// TwinCAT 3 PLC project RunTimeRoofControl
// Title: STELLA DachSteuerung
// Company: Leibniz Institut fuer Astrophysik Potsdam
// Author: J.Weingrill
// ProgramVersion: 3.1.4020.10
// libraries:
//   Tc2_Math, * (Beckhoff Automation GmbH)
//   Tc2_Standard, * (Beckhoff Automation GmbH)
//   Tc2_System, * (Beckhoff Automation GmbH)
//   Tc2_Utilities, * (Beckhoff Automation GmbH)
//   Tc3_IotBase, * (Beckhoff Automation GmbH)
//   Tc3_Module, * (Beckhoff Automation GmbH)
// project tree:
//   DUTs/ E_ErrorFlag.TcDUT, E_RoofCommand.TcDUT, E_RoofMode.TcDUT, E_RoofStatus.TcDUT
//   GVLs/ GVL_Environment.TcGVL, GVL_Infrastructure.TcGVL, GVL_Panel.TcGVL, GVL_Roof.TcGVL
//   / PlcTask.TcTTO
//   POUs/ Auxiliary.TcPOU, CalibrationUnit.TcPOU, Chamber.TcPOU, DehumidifierControl.TcPOU, Logging.TcPOU, MAIN.TcPOU, Environment.TcPOU
//   POUs/Function Blocks/ FB_AstroClock.TcPOU (not stored), FB_BLINK.TcPOU, FB_Dust.TcPOU (not stored), FB_EQ2HOR2.TcPOU (not stored), FB_EventLog.TcPOU, FB_Kalman1D.TcPOU, FB_MQTTCommunication.TcPOU, FB_PRECESS3.TcPOU, FB_RoofControl.TcPOU, FB_StatusLamp.TcPOU, FB_SUNPOS.TcPOU (not stored), FB_TimeAverage.TcPOU (not stored), InfluxMessage.TcPOU (not stored), LIGHT_BUTTON.TcPOU, TIMER.TcPOU
//   POUs/Functions/ APPEND.TcPOU (not stored), ATAN2.TcPOU (not stored), CT2LST.TcPOU (not stored), DateTime2JD.TcPOU (not stored), F_RainConversion.TcPOU (not stored), F_Y.TcPOU, Refraction.TcPOU (not stored), RoofStatus_TO_String.TcPOU
// real-time tasks:
//   TASK PlcTask: cycle T#10ms, priority 20, ADS port 350
// I/O:
//   DEVICE Device 1 (EtherCAT), AmsNetId 5.40.71.146.2.1
//     Term 1 (EK1200) [EK1200-5000 EtherCAT Power supply (2A E-Bus)]
//       Modul1 (EL2008) [EL2008 8Ch. Dig. Output 24V, 0.5A]
//       Modul2 (EL1008) [EL1008 8Ch. Dig. Input 24V, 3ms]
//       Modul3 (EL1008) [EL1008 8Ch. Dig. Input 24V, 3ms]
//       Modul4 (EL2008) [EL2008 8Ch. Dig. Output 24V, 0.5A]
//       Modul5 (EL1008) [EL1008 8Ch. Dig. Input 24V, 3ms]
//       Modul6 (EL1008) [EL1008 8Ch. Dig. Input 24V, 3ms] // Überstromkette Dach2
//       Modul7 (EL1008) [EL1008 8Ch. Dig. Input 24V, 3ms] // Panel
//       Modul8 (EL3068) [EL3068 8Ch. Ana. Input 0-10V] // Umweltsensoren innen
//       Modul9 (EL2008) [EL2008 8Ch. Dig. Output 24V, 0.5A]
//       Term 21 (EL9410) [EL9410 E-Bus Power Supplier  (Diagnostics)]
//       Modul10 (EL1024) [EL1024 4Ch. Dig. Input 24V, Type 2, 3ms] // Lichtschalter
//       Modul11 (EL3024) [EL3024 4Ch. Ana. Input 4-20mA DIFF]
//       Term 31 (EK1521) [EK1521 1 port EtherCAT junction (FX-MultiMode)]
//         WeatherStation1 (EK1501) [EK1501 EtherCAT Coupler (2A E-Bus, FX-MultiMode, ID switch)]
//           Term 33 (EL3068) [EL3068 8Ch. Ana. Input 0-10V]
//           Term 34 (EL1024) [EL1024 4Ch. Dig. Input 24V, Type 2, 3ms]
//           Term 35 (EL3024) [EL3024 4Ch. Ana. Input 4-20mA DIFF] // 1 Humidity,Temperature
//           Term 44 (EL6021) [EL6021 Interface (RS422/485)]
//           Term 41 (EL9011) [EL9011 End Terminal]
//       Term 36 (EK1521) [EK1521 1 port EtherCAT junction (FX-MultiMode)]
//         WeatherStation2 (EK1501) [EK1501 EtherCAT Coupler (2A E-Bus, FX-MultiMode, ID switch)]
//           Term 38 (EL3068) [EL3068 8Ch. Ana. Input 0-10V]
//           Term 39 (EL1024) [EL1024 4Ch. Dig. Input 24V, Type 2, 3ms]
//           Term 40 (EL3024) [EL3024 4Ch. Ana. Input 4-20mA DIFF]
//           Term 53 (EL6021) [EL6021 Interface (RS422/485)]
//           Term 42 (EL9011) [EL9011 End Terminal]
//       Term 56 (EK1521) [EK1521 1 port EtherCAT junction (FX-MultiMode)]
//         CalibrationUnit (EK1501) [EK1501 EtherCAT Coupler (2A E-Bus, FX-MultiMode, ID switch)]
//           Term 68 (EL1008) [EL1008 8Ch. Dig. Input 24V, 3ms]
//           Term 60 (EL2008) [EL2008 8Ch. Dig. Output 24V, 0.5A]
//           Term 61 (EL3164) [EL3164 4Ch. Ana. Input 0-10V]
//           Term 62 (EL3052) [EL3052 2Ch. Ana. Input 4-20mA]
//           Term 63 (EL3202-0010) [EL3202-0010 2Ch. Ana. Input PT100 (RTD), High Precision]
//           Term 64 (EL3202-0010) [EL3202-0010 2Ch. Ana. Input PT100 (RTD), High Precision]
//           Term 65 (EL3202-0010) [EL3202-0010 2Ch. Ana. Input PT100 (RTD), High Precision]
//           Term 76 (EK1110) [EK1110 EtherCAT extension]
//         Spectrograph Room (EK1100) [EK1100 EtherCAT Coupler (2A E-Bus)]
//           Term 79 (EL3202-0010) [EL3202-0010 2Ch. Ana. Input PT100 (RTD), High Precision]
//           Term 80 (EL3202-0010) [EL3202-0010 2Ch. Ana. Input PT100 (RTD), High Precision]
//           Term 81 (EL3202-0010) [EL3202-0010 2Ch. Ana. Input PT100 (RTD), High Precision]
//           Term 82 (EL3054) [EL3054 4Ch. Ana. Input 4-20mA]
//           Term 88 (EL9011) [EL9011 End Terminal]
//       Term 71 (EL9011) [EL9011 End Terminal]
//       Term 47 (EL9505) [EL9505 Power supply terminal 5V]
//       Term 48 (EL1124) [EL1124 4Ch. Dig. Input 5V, 10µs, Sensor Power]
//       Term 58 (EL1008) [EL1008 8Ch. Dig. Input 24V, 3ms]
//       Term 51 (EL9011) [EL9011 End Terminal]
//   DEVICE Device 3 (EtherCAT Automation Protocol) (disabled), AmsNetId 5.40.71.146.4.1
// variable links:
//   RunTimeRoofControl/RunTimeRoofControl Instance <-> Device 1 (EtherCAT)/Term 1 (EK1200)/Modul1 (EL2008)
//     PlcTask Outputs/GVL_Roof.ODach1Schnell <-> Channel 7/GVL_Roof.ODach1Schnell
//     PlcTask Outputs/GVL_Roof.ODach1auf <-> Channel 1/GVL_Roof.ODach1auf
//     PlcTask Outputs/GVL_Roof.ODach1zu <-> Channel 2/GVL_Roof.ODach1zu
//     PlcTask Outputs/GVL_Roof.ORiegel11auf <-> Channel 3/GVL_Roof.ORiegel11auf
//     PlcTask Outputs/GVL_Roof.ORiegel21auf <-> Channel 4/GVL_Roof.ORiegel21auf
//     PlcTask Outputs/GVL_Roof.ORiegel11zu <-> Channel 5/GVL_Roof.ORiegel11zu
//     PlcTask Outputs/GVL_Roof.ORiegel21zu <-> Channel 6/GVL_Roof.ORiegel21zu
//   RunTimeRoofControl/RunTimeRoofControl Instance <-> Device 1 (EtherCAT)/Term 1 (EK1200)/Modul10 (EL1024)
//     PlcTask Inputs/GVL_Environment.LightSwitch <-> Channel 1/Environment.LightSwitch
//   RunTimeRoofControl/RunTimeRoofControl Instance <-> Device 1 (EtherCAT)/Term 1 (EK1200)/Modul11 (EL3024)
//     PlcTask Inputs/GVL_Environment.DustSensorError <-> AI Standard Channel 1/Status/Error
//     PlcTask Inputs/GVL_Environment.rawDust <-> AI Standard Channel 1/Dust
//   RunTimeRoofControl/RunTimeRoofControl Instance <-> Device 1 (EtherCAT)/Term 1 (EK1200)/Modul2 (EL1008)
//     PlcTask Inputs/GVL_Roof.IDach1auf <-> Channel 1/GVL_Roof.IDach1auf
//     PlcTask Inputs/GVL_Roof.IDach1auf2 <-> Channel 2/GVL_Roof.IDach1auf2
//     PlcTask Inputs/GVL_Roof.IDach1zu <-> Channel 7/GVL_Roof.IDach1zu
//     PlcTask Inputs/GVL_Roof.IDach1zu2 <-> Channel 8/GVL_Roof.IDach1zu2
//     PlcTask Inputs/GVL_Roof.IRiegel11auf <-> Channel 3/GVL_Roof.IRiegel11auf
//     PlcTask Inputs/GVL_Roof.IRiegel21auf <-> Channel 4/GVL_Roof.IRiegel21auf
//     PlcTask Inputs/GVL_Roof.IRiegel11zu <-> Channel 5/GVL_Roof.IRiegel11zu
//     PlcTask Inputs/GVL_Roof.IRiegel21zu <-> Channel 6/GVL_Roof.IRiegel21zu
//   RunTimeRoofControl/RunTimeRoofControl Instance <-> Device 1 (EtherCAT)/Term 1 (EK1200)/Modul3 (EL1008)
//     PlcTask Inputs/GVL_Roof.IMotorschutz{11..16} <-> Channel {1..6}/GVL_Roof.IMotorschutz{11..16}  (6 links)
//   RunTimeRoofControl/RunTimeRoofControl Instance <-> Device 1 (EtherCAT)/Term 1 (EK1200)/Modul4 (EL2008)
//     PlcTask Outputs/GVL_Roof.ODach2Schnell <-> Channel 7/GVL_Roof.ODach2Schnell
//     PlcTask Outputs/GVL_Roof.ODach2auf <-> Channel 1/GVL_Roof.ODach2auf
//     PlcTask Outputs/GVL_Roof.ODach2zu <-> Channel 2/GVL_Roof.ODach2zu
//     PlcTask Outputs/GVL_Roof.ORiegel12auf <-> Channel 3/GVL_Roof.ORiegel12auf
//     PlcTask Outputs/GVL_Roof.ORiegel22auf <-> Channel 4/GVL_Roof.ORiegel22auf
//     PlcTask Outputs/GVL_Roof.ORiegel12zu <-> Channel 5/GVL_Roof.ORiegel12zu
//     PlcTask Outputs/GVL_Roof.ORiegel22zu <-> Channel 6/GVL_Roof.ORiegel22zu
//   RunTimeRoofControl/RunTimeRoofControl Instance <-> Device 1 (EtherCAT)/Term 1 (EK1200)/Modul5 (EL1008)
//     PlcTask Inputs/GVL_Roof.IDach2auf <-> Channel 1/GVL_Roof.IDach2auf
//     PlcTask Inputs/GVL_Roof.IDach2auf2 <-> Channel 2/GVL_Roof.IDach2auf2
//     PlcTask Inputs/GVL_Roof.IDach2zu <-> Channel 7/GVL_Roof.IDach2zu
//     PlcTask Inputs/GVL_Roof.IDach2zu2 <-> Channel 8/GVL_Roof.IDach2zu2
//     PlcTask Inputs/GVL_Roof.IRiegel12auf <-> Channel 3/GVL_Roof.IRiegel12auf
//     PlcTask Inputs/GVL_Roof.IRiegel22auf <-> Channel 4/GVL_Roof.IRiegel22auf
//     PlcTask Inputs/GVL_Roof.IRiegel12zu <-> Channel 5/GVL_Roof.IRiegel12zu
//     PlcTask Inputs/GVL_Roof.IRiegel22zu <-> Channel 6/GVL_Roof.IRiegel22zu
//   RunTimeRoofControl/RunTimeRoofControl Instance <-> Device 1 (EtherCAT)/Term 1 (EK1200)/Modul6 (EL1008)
//     PlcTask Inputs/GVL_Roof.IMotorschutz{21..26} <-> Channel {1..6}/GVL_Roof.IMotorschutz{21..26}  (6 links)
//   RunTimeRoofControl/RunTimeRoofControl Instance <-> Device 1 (EtherCAT)/Term 1 (EK1200)/Modul7 (EL1008)
//     PlcTask Inputs/GVL_Panel.ILeftCloseswitch <-> Channel 3/GVL_Panel.ILeftCloseswitch
//     PlcTask Inputs/GVL_Panel.ILeftOpenswitch <-> Channel 2/GVL_Panel.ILeftOpenswitch
//     PlcTask Inputs/GVL_Panel.IManualSwitch <-> Channel 1/GVL_Panel.IManualSwitch
//     PlcTask Inputs/GVL_Panel.IRightCloseSwitch <-> Channel 5/GVL_Panel.IRightCloseSwitch
//     PlcTask Inputs/GVL_Panel.IRightOpenSwitch <-> Channel 4/GVL_Panel.IRightOpenSwitch
//     PlcTask Inputs/GVL_Roof.IDach1Schnell <-> Channel 7/GVL_Roof.IDach1Schnell
//     PlcTask Inputs/GVL_Roof.IDach2Schnell <-> Channel 8/GVL_Roof.IDach2Schnell
//   RunTimeRoofControl/RunTimeRoofControl Instance <-> Device 1 (EtherCAT)/Term 1 (EK1200)/Modul8 (EL3068)
//     PlcTask Inputs/GVL_Environment.rawHumidityBay <-> AI Standard Channel 4/Environment.rawHumidityBay
//     PlcTask Inputs/GVL_Environment.rawHumidity_Electronics <-> AI Standard Channel 2/Environment.rawHumidity_Electronics
//     PlcTask Inputs/GVL_Environment.rawHumidity_Spec <-> AI Standard Channel 6/Environment.rawHumidity_Spec
//     PlcTask Inputs/GVL_Environment.rawPressureBay <-> AI Standard Channel 8/GVL_Environment.rawPressureBay
//     PlcTask Inputs/GVL_Environment.rawTemperatureBay <-> AI Standard Channel 3/Environment.rawTemperatureBay
//     PlcTask Inputs/GVL_Environment.rawTemperature_Electronics <-> AI Standard Channel 1/Environment.rawTemperature_Electronics
//     PlcTask Inputs/GVL_Environment.rawTemperature_Spec <-> AI Standard Channel 5/Environment.rawTemperature_Spec
//     PlcTask Inputs/GVL_Environment.rawWindSpeedBay <-> AI Standard Channel 7/Environment.rawWindSpeedBay
//   RunTimeRoofControl/RunTimeRoofControl Instance <-> Device 1 (EtherCAT)/Term 1 (EK1200)/Modul9 (EL2008)
//     PlcTask Outputs/GVL_Environment.Dehumidifier <-> Channel 4/Environment.Dehumidifier
//     PlcTask Outputs/GVL_Environment.Horn <-> Channel 3/Environment.Horn
//     PlcTask Outputs/GVL_Environment.LightBay <-> Channel 1/Environment.LightBay
//     PlcTask Outputs/GVL_Environment.RoofPower <-> Channel 2/Environment.RoofPower
//     PlcTask Outputs/GVL_Panel.Roof1Lamp <-> Channel 7/GVL_Panel.Roof1Lamp
//     PlcTask Outputs/GVL_Panel.Roof2Lamp <-> Channel 8/GVL_Panel.Roof2Lamp
//   RunTimeRoofControl/RunTimeRoofControl Instance <-> Device 1 (EtherCAT)/Term 1 (EK1200)/Term 21 (EL9410)
//     PlcTask Inputs/GVL_Panel.Up_Undervoltage <-> Status Up/Undervoltage
//     PlcTask Inputs/GVL_Panel.Us_Undervoltage <-> Status Us/Undervoltage
//   RunTimeRoofControl/RunTimeRoofControl Instance <-> Device 1 (EtherCAT)/Term 1 (EK1200)/Term 31 (EK1521)/WeatherStation1 (EK1501)/Term 33 (EL3068)
//     PlcTask Inputs/GVL_Environment.rawBrightness1 <-> AI Standard Channel 2/GVL_Environment.rawBrightness1
//     PlcTask Inputs/GVL_Environment.rawHumidity1 <-> AI Standard Channel 4/GVL_Environment.rawHumidity1
//     PlcTask Inputs/GVL_Environment.rawLightDirection <-> AI Standard Channel 1/GVL_Environment.rawLightDirection
//     PlcTask Inputs/GVL_Environment.rawPressure <-> AI Standard Channel 3/GVL_Environment.rawPressure
//     PlcTask Inputs/GVL_Environment.rawRain_analogue1 <-> AI Standard Channel 6/GVL_Environment.rawRain_analogue1
//     PlcTask Inputs/GVL_Environment.rawTemperature1 <-> AI Standard Channel 5/GVL_Environment.rawTemperature1
//     PlcTask Inputs/GVL_Environment.rawWindDirection <-> AI Standard Channel 7/GVL_Environment.rawWindDirection
//     PlcTask Inputs/GVL_Environment.rawWindSpeed1 <-> AI Standard Channel 8/GVL_Environment.rawWindSpeed1
//   RunTimeRoofControl/RunTimeRoofControl Instance <-> Device 1 (EtherCAT)/Term 1 (EK1200)/Term 31 (EK1521)/WeatherStation1 (EK1501)/Term 34 (EL1024)
//     PlcTask Inputs/GVL_Environment.Rain_alarm1 <-> Channel 1/Environment.Rain_alarm1
//   RunTimeRoofControl/RunTimeRoofControl Instance <-> Device 1 (EtherCAT)/Term 1 (EK1200)/Term 36 (EK1521)/WeatherStation2 (EK1501)/Term 38 (EL3068)
//     PlcTask Inputs/GVL_Environment.rawBrightness <-> AI Standard Channel 4/Environment.rawBrightness
//     PlcTask Inputs/GVL_Environment.rawBrightnessLow <-> AI Standard Channel 5/Environment.rawBrightnessLow
//     PlcTask Inputs/GVL_Environment.rawHumidity2 <-> AI Standard Channel 2/Environment.rawHumidity2
//     PlcTask Inputs/GVL_Environment.rawTemperature2 <-> AI Standard Channel 3/Environment.rawTemperature2
//     PlcTask Inputs/GVL_Environment.rawWindSpeed2 <-> AI Standard Channel 1/Environment.rawWindSpeed2
//   RunTimeRoofControl/RunTimeRoofControl Instance <-> Device 1 (EtherCAT)/Term 1 (EK1200)/Term 36 (EK1521)/WeatherStation2 (EK1501)/Term 39 (EL1024)
//     PlcTask Inputs/GVL_Environment.Rain_alarm2 <-> Channel 1/Environment.Rain_alarm2
//   RunTimeRoofControl/RunTimeRoofControl Instance <-> Device 1 (EtherCAT)/Term 1 (EK1200)/Term 48 (EL1124)
//     PlcTask Inputs/GVL_Environment.rawDust11 <-> Channel 1/Environment.rawDust11
//     PlcTask Inputs/GVL_Environment.rawDust12 <-> Channel 2/Environment.rawDust12
//     PlcTask Inputs/GVL_Environment.rawDust21 <-> Channel 3/Environment.rawDust21
//     PlcTask Inputs/GVL_Environment.rawDust22 <-> Channel 4/Environment.rawDust22
//   RunTimeRoofControl/RunTimeRoofControl Instance <-> Device 1 (EtherCAT)/Term 1 (EK1200)/Term 56 (EK1521)/CalibrationUnit (EK1501)/Term 60 (EL2008)
//     PlcTask Outputs/CalibrationUnit.Halolamp1 <-> Channel 3/CalibrationUnit.Halolamp1
//     PlcTask Outputs/CalibrationUnit.Halolamp2 <-> Channel 4/CalibrationUnit.Halolamp2
//     PlcTask Outputs/CalibrationUnit.ThArlamp1 <-> Channel 1/CalibrationUnit.ThArlamp1
//     PlcTask Outputs/CalibrationUnit.ThArlamp2 <-> Channel 2/CalibrationUnit.ThArlamp2
//   RunTimeRoofControl/RunTimeRoofControl Instance <-> Device 1 (EtherCAT)/Term 1 (EK1200)/Term 56 (EK1521)/CalibrationUnit (EK1501)/Term 61 (EL3164)
//     PlcTask Inputs/CalibrationUnit.SESdewarpressureraw <-> AI Standard Channel 1/CalibrationUnit.SESdewarpressureraw
//     PlcTask Inputs/CalibrationUnit.SESpumppressureraw <-> AI Standard Channel 2/CalibrationUnit.SESpumppressureraw
//   RunTimeRoofControl/RunTimeRoofControl Instance <-> Device 1 (EtherCAT)/Term 1 (EK1200)/Term 56 (EK1521)/CalibrationUnit (EK1501)/Term 62 (EL3052)
//     PlcTask Inputs/CalibrationUnit.cryoreturnraw <-> AI Standard Channel 1/CalibrationUnit.cryoreturnraw
//     PlcTask Inputs/CalibrationUnit.cryosupplyraw <-> AI Standard Channel 2/CalibrationUnit.cryosupplyraw
//   RunTimeRoofControl/RunTimeRoofControl Instance <-> Device 1 (EtherCAT)/Term 1 (EK1200)/Term 56 (EK1521)/CalibrationUnit (EK1501)/Term 63 (EL3202-0010)
//     PlcTask Inputs/CalibrationUnit.rawTemperature1 <-> RTD Inputs Channel 1/CalibrationUnit.rawTemperature1
//     PlcTask Inputs/CalibrationUnit.rawTemperature2 <-> RTD Inputs Channel 2/CalibrationUnit.rawTemperature2
//   RunTimeRoofControl/RunTimeRoofControl Instance <-> Device 1 (EtherCAT)/Term 1 (EK1200)/Term 56 (EK1521)/CalibrationUnit (EK1501)/Term 64 (EL3202-0010)
//     PlcTask Inputs/CalibrationUnit.rawTemperature3 <-> RTD Inputs Channel 1/CalibrationUnit.rawTemperature3
//     PlcTask Inputs/CalibrationUnit.rawTemperature4 <-> RTD Inputs Channel 2/CalibrationUnit.rawTemperature4
//   RunTimeRoofControl/RunTimeRoofControl Instance <-> Device 1 (EtherCAT)/Term 1 (EK1200)/Term 56 (EK1521)/CalibrationUnit (EK1501)/Term 65 (EL3202-0010)
//     PlcTask Inputs/CalibrationUnit.rawTemperature5 <-> RTD Inputs Channel 1/CalibrationUnit.rawTemperature5
//     PlcTask Inputs/CalibrationUnit.rawTemperature6 <-> RTD Inputs Channel 2/CalibrationUnit.rawTemperature6
//   RunTimeRoofControl/RunTimeRoofControl Instance <-> Device 1 (EtherCAT)/Term 1 (EK1200)/Term 56 (EK1521)/CalibrationUnit (EK1501)/Term 68 (EL1008)
//     PlcTask Inputs/CalibrationUnit.lampsensor1 <-> Channel 1/CalibrationUnit.lampsensor1
//     PlcTask Inputs/CalibrationUnit.lampsensor2 <-> Channel 2/CalibrationUnit.lampsensor2
//   RunTimeRoofControl/RunTimeRoofControl Instance <-> Device 1 (EtherCAT)/Term 1 (EK1200)/Term 56 (EK1521)/Spectrograph Room (EK1100)/Term 79 (EL3202-0010)
//     PlcTask Inputs/Chamber.rawTemperature1 <-> RTD Inputs Channel 1/Chamber.rawTemperature1
//     PlcTask Inputs/Chamber.rawTemperature2 <-> RTD Inputs Channel 2/Chamber.rawTemperature2
//   RunTimeRoofControl/RunTimeRoofControl Instance <-> Device 1 (EtherCAT)/Term 1 (EK1200)/Term 56 (EK1521)/Spectrograph Room (EK1100)/Term 80 (EL3202-0010)
//     PlcTask Inputs/Chamber.rawTemperature3 <-> RTD Inputs Channel 1/Chamber.rawTemperature3
//     PlcTask Inputs/Chamber.rawTemperature4 <-> RTD Inputs Channel 2/Chamber.rawTemperature4
//   RunTimeRoofControl/RunTimeRoofControl Instance <-> Device 1 (EtherCAT)/Term 1 (EK1200)/Term 56 (EK1521)/Spectrograph Room (EK1100)/Term 81 (EL3202-0010)
//     PlcTask Inputs/Chamber.rawTemperature5 <-> RTD Inputs Channel 1/Value
//     PlcTask Inputs/Chamber.rawTemperature6 <-> RTD Inputs Channel 2/Value
//   RunTimeRoofControl/RunTimeRoofControl Instance <-> Device 1 (EtherCAT)/Term 1 (EK1200)/Term 56 (EK1521)/Spectrograph Room (EK1100)/Term 82 (EL3054)
//     PlcTask Inputs/Chamber.rawpressure <-> AI Standard Channel 1/Chamber.rawpressure
//   RunTimeRoofControl/RunTimeRoofControl Instance <-> Device 1 (EtherCAT)/Term 1 (EK1200)/Term 58 (EL1008)
//     PlcTask Inputs/GVL_Infrastructure.MainUPS_BatteryLow <-> Channel 3/GVL_Infrastructure.MainUPS_BatteryLow
//     PlcTask Inputs/GVL_Infrastructure.MainUPS_CommonAlarm <-> Channel 4/GVL_Infrastructure.MainUPS_CommonAlarm
//     PlcTask Inputs/GVL_Infrastructure.MainUPS_LoadOnInverter <-> Channel 2/GVL_Infrastructure.MainUPS_LoadOnInverter
//     PlcTask Inputs/GVL_Infrastructure.MainUPS_MainsPreset <-> Channel 1/GVL_Infrastructure.MainUPS_MainsPreset

CONFIGURATION RunTimeRoofControl
    RESOURCE PLC ON TwinCAT3
        TASK PlcTask(INTERVAL := T#10ms, PRIORITY := 20);
        PROGRAM MAIN WITH PlcTask : MAIN;
    END_RESOURCE
END_CONFIGURATION

// ---- DUTs/E_ErrorFlag.TcDUT
{attribute 'qualified_only'}
{attribute 'strict'}
TYPE E_ErrorFlag :
(
	noError := 0,
	ErrorOneLocked,
	ErrorNotUnlocked,
	ErrorLockUnlock,
	ErrorOpenClose,
	ErrorOpenLocked
);
END_TYPE

// ---- DUTs/E_RoofCommand.TcDUT
TYPE E_RoofCommand :
(
	CloseRoof,
 	OpenRoof,
	StopRoof
);
END_TYPE

// ---- DUTs/E_RoofMode.TcDUT
TYPE E_RoofMode :
(
	RoofAutomatic := 0,
 	RoofManual := 1
);
END_TYPE

// ---- DUTs/E_RoofStatus.TcDUT
TYPE E_RoofStatus :
(
	StatusUndefined 	:= 0,
	StatusClosed 		:= 100,
	StatusLocking 		:= 200,
	StatusLocked 		:= 300,
	StatusUnlocking 	:= 400,
	StatusUnlocked 		:= 500,
	StatusStartOpening 	:= 600,
	StatusOpening 		:= 700,
	StatusEndOpening 	:= 800,
	StatusOpened 		:= 900,
	StatusStartClosing 	:= 1000,
	StatusClosing 		:= 1100,
	StatusEndClosing 	:= 1200,
	
	StatusError 		:= -1
);
END_TYPE

// ---- GVLs/GVL_Environment.TcGVL
{attribute 'qualified_only'}

(* 
source: sensors-upgrade.pdf
STELLA building control sensors & switches 
*)

VAR_GLOBAL
		
	// Weather Station 1
	rawLightDirection			AT%I*:	INT;
	rawBrightness1				AT%I*:	INT;
	rawPressure 				AT%I*:	INT;
	rawHumidity1				AT%I*:	INT;
	rawTemperature1				AT%I*:	INT;
	rawRain_analogue1			AT%I*:	INT;
	rawWindDirection			AT%I*:	INT;
	Rain_alarm1					AT%I*:	BOOL;
	rawWindSpeed1				AT%I*:	INT;
	Overcorrect_status1			AT%I*:	BOOL;
	
	// Weather Station 2
	rawWindSpeed2				AT%I*:	INT;
	rawTemperature2				AT%I*:	INT;
	rawHumidity2				AT%I*:	INT;
	Rain_alarm2					AT%I*:	BOOL;
	rawBrightness				AT%I*:	INT;
	rawBrightnessLow			AT%I*:	INT;
	Overcorrect_status2			AT%I*:	BOOL;

	// indoors
	rawTemperature_Electronics	AT%I*:	INT;
	rawHumidity_Electronics		AT%I*:	INT;
	rawTemperatureBay			AT%I*:	INT;
	rawHumidityBay				AT%I*:	INT;
	rawTemperature_Spec			AT%I*:	INT;
	rawHumidity_Spec			AT%I*:	INT;
	
	// Bay
	rawWindSpeedBay				AT%I*:	INT;
	rawPressureBay 				AT%I*:	INT;
	// Dust Sensor 4..20mA
	rawDust						AT%I*:	INT;

	// Horn für Warnung beim Öffnen und Schliessen
	Horn						AT%Q*:	BOOL;
	// Entfeuchter
	Dehumidifier				AT%Q*:	BOOL;
	// RoofPower
	RoofPower					AT%Q*:	BOOL;
	// Licht in der Kuppel an
	LightBay					AT%Q*:	BOOL;

	// Lichtschalter in der Kuppel
	LightSwitch					AT%I*:	BOOL;
	
	// sensor error
	DustSensorError				AT%I*:	BOOL;
	rawDust11					AT%I*:	BOOL;
	rawDust12					AT%I*:	BOOL;
	rawDust21					AT%I*:	BOOL;
	rawDust22					AT%I*:	BOOL;
	
	//rawDust22: INT;
END_VAR

// ---- GVLs/GVL_Infrastructure.TcGVL
{attribute 'qualified_only'}
VAR_GLOBAL
	MainUPS_MainsPreset		AT%I*:	BOOL;
	MainUPS_LoadOnInverter		AT%I*:	BOOL;
	MainUPS_BatteryLow		AT%I*:	BOOL;
	MainUPS_CommonAlarm		AT%I*:	BOOL;

END_VAR

// ---- GVLs/GVL_Panel.TcGVL
{attribute 'qualified_only'}
VAR_GLOBAL
	// switch between automatic and manul
	IManualSwitch		AT%I*:	BOOL;
	// left open switch
	ILeftOpenswitch		AT%I*:	BOOL;
	// left close switch
	ILeftCloseswitch	AT%I*:	BOOL;
	// right open switch
	IRightOpenSwitch	AT%I*:	BOOL;
	// right close switch
	IRightCloseSwitch	AT%I*:	BOOL;
	
	// roof status lamp 1	
	Roof1Lamp			AT%Q*:	BOOL;
	// roof status lamp 2
	Roof2Lamp			AT%Q*:	BOOL;
	//EL9410 status US
	Us_Undervoltage		AT%I*:	BOOL;
	//EL9410 status Up
	Up_Undervoltage		AT%I*:	BOOL;
END_VAR

// ---- GVLs/GVL_Roof.TcGVL
{attribute 'qualified_only'}
VAR_GLOBAL
	//KDach1auf
	IDach1auf		AT%I*:	BOOL;
	//KDach1auf2
	IDach1auf2		AT%I*:	BOOL;
	//KDach1zu
	IDach1zu		AT%I*:	BOOL;
	//KDach1zu2
	IDach1zu2		AT%I*:	BOOL;
	//KRiegel11auf
	IRiegel11auf	AT%I*:	BOOL;
	//KRiegel12auf
	IRiegel21auf	AT%I*:	BOOL;
	//KRiegel11zu
	IRiegel11zu		AT%I*:	BOOL;
	//KRiegel12zu
	IRiegel21zu		AT%I*:	BOOL;
	//KDach1schnell
	IDach1Schnell	AT%I*:	BOOL;
	// MS1NC1
	IMotorschutz11	AT%I*:	BOOL;
	// MS2NC1
	IMotorschutz12	AT%I*:	BOOL;
	// MS3NC1
	IMotorschutz13	AT%I*:	BOOL;
	// MS4NC1
	IMotorschutz14	AT%I*:	BOOL;
	// MS5NC1
	IMotorschutz15	AT%I*:	BOOL;
	// MS6NC1
	IMotorschutz16	AT%I*:	BOOL;

	IDach2auf		AT%I*:	BOOL;
	IDach2auf2		AT%I*:	BOOL;
	IDach2zu		AT%I*:	BOOL;
	IDach2zu2		AT%I*:	BOOL;
	IRiegel12auf	AT%I*:	BOOL;
	IRiegel22auf	AT%I*:	BOOL;
	IRiegel12zu		AT%I*:	BOOL;
	IRiegel22zu		AT%I*:	BOOL;
	IDach2Schnell	AT%I*:	BOOL;
	//MS1NC2
	IMotorschutz21	AT%I*:	BOOL;
	//MS2NC2
	IMotorschutz22	AT%I*:	BOOL;
	//MS3NC2
	IMotorschutz23	AT%I*:	BOOL;
	//MS4NC2
	IMotorschutz24	AT%I*:	BOOL;
	//MS5NC2
	IMotorschutz25	AT%I*:	BOOL;
	//MS6NC2
	IMotorschutz26	AT%I*:	BOOL;
	
	// Dig. Output
	ODach1auf		AT%Q*:	BOOL;
	ODach1zu		AT%Q*:	BOOL;
	ORiegel11auf	AT%Q*:	BOOL;
	ORiegel21auf	AT%Q*:	BOOL;
	ORiegel11zu		AT%Q*:	BOOL;
	ORiegel21zu		AT%Q*:	BOOL;
	ODach1Schnell	AT%Q*:	BOOL;

	ODach2auf		AT%Q*:	BOOL;
	ODach2zu		AT%Q*:	BOOL;
	ORiegel12auf	AT%Q*:	BOOL;
	ORiegel22auf	AT%Q*:	BOOL;
	ORiegel12zu		AT%Q*:	BOOL;
	ORiegel22zu		AT%Q*:	BOOL;
	ODach2Schnell	AT%Q*:	BOOL;
	
END_VAR

// ---- POUs/MAIN.TcPOU
PROGRAM MAIN
VAR_INPUT
	// open the roof remotely
	OpenRoofAuto: 	BOOL;
	// close the roof remotely
	CloseRoofAuto: 	BOOL;
	// stop the roof remotely (unused?)
	StopRoofAuto: 	BOOL;
	// turn on the light remotely
	LightAuto: 		BOOL;
END_VAR

VAR
	// RoofManual or RoofAutomatic
	nMode:		    E_RoofMode;
	// DachControl roof1
	Dach1Control:	FB_RoofControl;
	// DachControl roof 2
	Dach2Control:	FB_RoofControl;
	Roof1Command,
	Roof2Command:	E_RoofCommand;
	Roof1Status,
	Roof2Status,
	LastRoof1Status,
	LastRoof2Status:	E_RoofStatus;
	RSOpenRoof1,
	RSCloseRoof1,
	RSOpenRoof2,
	RSCloseRoof2: 	RS;
	OpenRoofAutoPending: BOOL;
	OpenRoof1,
	CloseRoof1,
	OpenRoof2,
	CloseRoof2,
	StopRoof1,
	StopRoof2:	BOOL;
	// report manual operation of the dome to TCS
	isRoofManual: BOOL;
	// indicates an error in the dust sensor
	DustSensorError: BOOL;
	// Timer for Dome Light
	LightTimer:		LIGHT_BUTTON;
	LightAutoTimer:	TP;
	RoofStatusLamp1,
	RoofStatusLamp2: FB_StatusLamp;
	WeatherAlarm,
	MotionAlarm1,
	MotionAlarm2:	BOOL;
	// indicates at least on environment signal is bad
	EnvironmentBad,
	// environment signal is bad for n seconds
	EnvironmentAlarm: BOOL;
	// time function block for Environment signal
	EnvironmentBadTimer: TON;
	MQTTTimer : TON := (PT:=T#5S);
	// MQTT class for publishing
	MQTTClient:		FB_MQTTCommunication;
	// precise astronomical	time
	fbTime: FB_AstroClock;
	// current Julian Date calculated from system time
	jd:				LREAL;
	// calculation for solar position
	sunpos:	FB_SUNPOS;
	eq2hor2: FB_EQ2HOR2;
	// Humidity Trigger
	HumidityTrigger:	SR;
	Roof1OpenTimer,
	Roof2OpenTimer,
	Roof1CloseTimer,
	Roof2CloseTimer:	TIMER;
	Roof1OpenTimeOut,
	Roof2OpenTimeOut,
	Roof1CloseTimeOut,
	Roof2CloseTimeOut:	TON;
	Roof1LockTimeOut,
	Roof2LockTimeOut,
	Roof1UnlockTimeOut,
	Roof2UnlockTimeOut:	TON;
	
	Roof1StatusWord:	WORD;
	Roof2StatusWord:	WORD;
END_VAR
VAR CONSTANT
	// telescope site longitude, source: Google 
	longitude: 		LREAL := -16.50926; //13.101867;
	// telescope site latitude, source: Google
	latitude: 		LREAL := 28.30120; //52.404940;

	HumidityLimitCritical:		REAL := 80.0;
	HumidityLimitHigh:		REAL := 75.0;
	HumidityLimitLow:		REAL := 55.0;
	
	WindSpeedLimit:		REAL := 20.0;
	WindSpeedBayLimit:	REAL :=	15.0;
	DustLimit:			REAL := 0.01;
	BrightnessLimit:	REAL := 40000.0;
END_VAR

IF GVL_Panel.IManualSwitch THEN
	nMode := RoofManual;
ELSE
	nMode := RoofAutomatic;
END_IF
isRoofManual := GVL_Panel.IManualSwitch;

DustSensorError := GVL_Environment.DustSensorError;

// initialize MQTT Communication
MQTTClient();

// collect weather data
Environment();

// Handle Auxiliary inputs and outputs
Auxiliary();

CalibrationUnit();
Chamber();

// Handle Logging
Logging();

// Control Logic for Dehumidifier
DehumidifierControl(Enable := nMode = RoofAutomatic AND Roof1Status = StatusLocked AND Roof2Status = StatusLocked);

HumidityTrigger(SET1 := Environment.Humidity >= HumidityLimitHigh,
				RESET := Environment.Humidity < HumidityLimitLow);

fbTime();
jd := DateTime2JD(fbTime.time_RTCEX2);
				
sunpos(JD := jd);
eq2hor2(alpha := sunpos.RA, delta := sunpos.Dec, lon := longitude, lat := latitude, JD := jd);
						
// define bad weather condition; rain is handled in EnvironmentAlarm
EnvironmentBad := (Environment.DustTrigger.Q1 AND NOT DustSensorError) OR
		HumidityTrigger.Q1 OR
		Environment.WindSpeed1 > WindSpeedLimit OR
		Environment.WindSpeed2 > WindSpeedLimit OR
		Environment.Windspeed_bay > WindSpeedBayLimit OR
		Environment.Brightness1 > BrightnessLimit OR 
		eq2hor2.alt > 6.0;

EnvironmentBadTimer(IN := EnvironmentBad,
					PT := T#125S);
					
EnvironmentAlarm := EnvironmentBadTimer.Q OR Environment.RainMasterAlarm;

IF nMode = RoofAutomatic THEN
	// if we get the open comand during bad weather, postpone the signal
	IF OpenRoofAuto AND EnvironmentAlarm THEN
		OpenRoofAutoPending := TRUE;
		OpenRoofAuto := FALSE;
	// if we get the close command cancle the signal
	ELSIF CloseRoofAuto THEN
		OpenRoofAutoPending := FALSE;
	END_IF
	// if weather is good, execute the pending signal
	IF NOT EnvironmentAlarm AND OpenRoofAutoPending THEN
		OpenRoofAuto := TRUE;
		OpenRoofAutoPending := FALSE;
	END_IF			
	
	IF CloseRoofAuto THEN
		OpenRoofAuto := FALSE;
		Roof1Command := CloseRoof;
		Roof2Command := CloseRoof;
	ELSIF OpenRoofAuto THEN
		CloseRoofAuto := FALSE;
		Roof1Command := OpenRoof;
		Roof2Command := OpenRoof;
	ELSE
		Roof1Command := StopRoof;
		Roof2Command := StopRoof;
	END_IF

	// overwrite previous command if the weather is bad for xx seconds
	IF EnvironmentAlarm THEN
		IF NOT (Roof1Status = StatusLocked) THEN
			Roof1Command := CloseRoof;	
		END_IF
		IF NOT (Roof2Status = StatusLocked) THEN
			Roof2Command := CloseRoof;	
		END_IF
	END_IF
	
	IF (Roof1Status = StatusLocked) AND (Roof2Status = StatusLocked) THEN
		CloseRoofAuto := FALSE;
	END_IF			
	IF (Roof1Status = StatusOpened) AND (Roof2Status = StatusOpened) THEN
		OpenRoofAuto := FALSE;
	END_IF			
	
ELSE //	RoofManual
	OpenRoof1 := GVL_Panel.ILeftOpenSwitch AND NOT GVL_Panel.ILeftCloseSwitch;
	CloseRoof1 := GVL_Panel.ILeftCloseSwitch AND NOT GVL_Panel.ILeftOpenSwitch;
	StopRoof1 := NOT (GVL_Panel.ILeftOpenSwitch XOR GVL_Panel.ILeftCloseSwitch);
	
	IF CloseRoof1 THEN
		Roof1Command := CloseRoof;
	ELSIF OpenRoof1 THEN
		Roof1Command := OpenRoof;
	ELSE
		Roof1Command := StopRoof;
	END_IF

	OpenRoof2 := GVL_Panel.IRightOpenSwitch AND NOT GVL_Panel.IRightCloseSwitch;
	CloseRoof2 := GVL_Panel.IRightCloseSwitch AND NOT GVL_Panel.IRightOpenSwitch;
	StopRoof2 := NOT (GVL_Panel.IRightOpenSwitch XOR GVL_Panel.IRightCloseSwitch);
	
	IF CloseRoof2 THEN
		Roof2Command := CloseRoof;
	ELSIF OpenRoof2 THEN
		Roof2Command := OpenRoof;
	ELSE
		Roof2Command := StopRoof;
	END_IF
	Weatheralarm := ((Roof1Status = StatusOpened) OR (Roof2Status = StatusOpened))
					AND EnvironmentAlarm;
		
END_IF

Roof1OpenTimer(bStart := (Roof1Command = OpenRoof) AND NOT (Roof1Status = StatusOpened));
Roof2OpenTimer(bStart := (Roof2Command = OpenRoof) AND NOT (Roof2Status = StatusOpened));
Roof1CloseTimer(bStart := (Roof1Command = CloseRoof) AND NOT (Roof1Status = StatusLocked));
Roof2CloseTimer(bStart := (Roof2Command = CloseRoof) AND NOT (Roof2Status = StatusLocked));

Roof1OpenTimeOut(IN := (Roof1Command = OpenRoof) AND NOT (Roof1Status = StatusOpened), PT := T#130S);
Roof2OpenTimeOut(IN := (Roof2Command = OpenRoof) AND NOT (Roof2Status = StatusOpened), PT := T#130S);
Roof1CloseTimeOut(IN := (Roof1Command = CloseRoof) AND NOT (Roof1Status = StatusLocked), PT := T#130S);
Roof2CloseTimeOut(IN := (Roof1Command = CloseRoof) AND NOT (Roof2Status = StatusLocked), PT := T#130S);

Roof1LockTimeOut(IN := (GVL_Roof.ORiegel11zu OR GVL_Roof.ORiegel21zu) AND NOT (GVL_Roof.IRiegel11zu OR GVL_Roof.IRiegel21zu), PT := T#10S);
Roof2LockTimeOut(IN := (GVL_Roof.ORiegel12zu OR GVL_Roof.ORiegel22zu) AND NOT (GVL_Roof.IRiegel12zu OR GVL_Roof.IRiegel22zu), PT := T#10S);

Roof1UnlockTimeOut(IN := (GVL_Roof.ORiegel11auf OR GVL_Roof.ORiegel21auf) AND NOT (GVL_Roof.IRiegel11auf OR GVL_Roof.IRiegel21auf), PT := T#10S);
Roof2UnlockTimeOut(IN := (GVL_Roof.ORiegel12auf OR GVL_Roof.ORiegel22auf) AND NOT (GVL_Roof.IRiegel12auf OR GVL_Roof.IRiegel22auf), PT := T#10S);

	
LightTimer( IN := GVL_Environment.LightSwitch, PT := T#1H);

// disable light after 15 minutes if on automatic			
LightAutoTimer(IN := LightAuto, PT := T#15M);

// automatic, manual on
IF nMode = RoofAutomatic THEN
	LightTimer.PT := T#1H;
	GVL_Environment.LightBay := LightTimer.Q OR (LightAutoTimer.Q AND LightAuto);
ELSIF nMode = RoofManual THEN
	LightTimer.PT := T#8H; // we are in service mode
	GVL_Environment.LightBay := LightTimer.Q;
ELSE
	GVL_Environment.LightBay := FALSE;
END_IF
IF (Roof1Status = StatusOpened) OR (Roof2Status = StatusOpened) THEN
	GVL_Environment.LightBay := FALSE;
END_IF


(*** Control Section ***)	

Dach1Control(   cmdRoofCommand := Roof1Command,
				bOpenSwitch1   := GVL_Roof.IDach1auf,
				bOpenSwitch2   := GVL_Roof.IDach1auf2,
				bClosedSwitch1 := GVL_Roof.IDach1zu,
				bClosedSwitch2 := GVL_Roof.IDach1zu2,
				bLocked1       := GVL_Roof.IRiegel11zu,
				bUnlocked1     := GVL_Roof.IRiegel11auf,
				bLocked2       := GVL_Roof.IRiegel21zu,
				bUnlocked2     := GVL_Roof.IRiegel21auf,
				bFastSwitch    := GVL_Roof.IDach1Schnell,
				bOpenLock1     => GVL_Roof.ORiegel11auf,
				bCloseLock1    => GVL_Roof.ORiegel11zu,
				bOpenLock2     => GVL_Roof.ORiegel21auf,
				bCloseLock2    => GVL_Roof.ORiegel21zu,
				bRoofOpen 	   => GVL_Roof.ODach1auf,
				bRoofClose     => GVL_Roof.ODach1zu,
				bMotorFast     => GVL_Roof.ODach1Schnell,
				RoofStatus     => Roof1Status,
				MotionAlarm    => MotionAlarm1);

Dach2Control(   cmdRoofCommand := Roof2Command,
				bOpenSwitch1   := GVL_Roof.IDach2auf,
				bOpenSwitch2   := GVL_Roof.IDach2auf2,
				bClosedSwitch1 := GVL_Roof.IDach2zu,
				bClosedSwitch2 := GVL_Roof.IDach2zu2,
				bLocked1       := GVL_Roof.IRiegel12zu,
				bUnlocked1     := GVL_Roof.IRiegel12auf,
				bLocked2       := GVL_Roof.IRiegel22zu,
				bUnlocked2     := GVL_Roof.IRiegel22auf,
				bFastSwitch    := GVL_Roof.IDach2Schnell,
				bOpenLock1     => GVL_Roof.ORiegel12auf,
				bCloseLock1    => GVL_Roof.ORiegel12zu,
				bOpenLock2     => GVL_Roof.ORiegel22auf,
				bCloseLock2    => GVL_Roof.ORiegel22zu,
				bRoofOpen      => GVL_Roof.ODach2auf,
				bRoofClose     => GVL_Roof.ODach2zu,
				bMotorFast     => GVL_Roof.ODach2Schnell,
				RoofStatus     => Roof2Status,
				MotionAlarm    => MotionAlarm2);


// Set status lamps
RoofStatusLamp1(RoofStatus := Roof1Status, RoofLamp => GVL_Panel.Roof1Lamp);
RoofStatusLamp2(RoofStatus := Roof2Status, RoofLamp => GVL_Panel.Roof2Lamp);
			
// sound horn
GVL_Environment.Horn := WeatherAlarm OR MotionAlarm1 OR MotionAlarm2;		

IF GVL_Panel.Us_Undervoltage OR GVL_Panel.Up_Undervoltage THEN
	Roof1Status := StatusError;
	Roof2Status := StatusError;
END_IF

// set status words
Roof1StatusWord.0   := GVL_Roof.IDach1auf;
Roof1StatusWord.1   := GVL_Roof.IDach1auf2;
Roof1StatusWord.2 	:= GVL_Roof.IDach1zu;
Roof1StatusWord.3 	:= GVL_Roof.IDach1zu2;
Roof1StatusWord.4   := GVL_Roof.IRiegel11zu;
Roof1StatusWord.5   := GVL_Roof.IRiegel11auf;
Roof1StatusWord.6   := GVL_Roof.IRiegel21zu;
Roof1StatusWord.7   := GVL_Roof.IRiegel21auf;
Roof1StatusWord.8   := GVL_Roof.IDach1Schnell;

Roof2StatusWord.0   := GVL_Roof.IDach2auf;
Roof2StatusWord.1   := GVL_Roof.IDach2auf2;
Roof2StatusWord.2 	:= GVL_Roof.IDach2zu;
Roof2StatusWord.3 	:= GVL_Roof.IDach2zu2;
Roof2StatusWord.4   := GVL_Roof.IRiegel12zu;
Roof2StatusWord.5   := GVL_Roof.IRiegel12auf;
Roof2StatusWord.6   := GVL_Roof.IRiegel22zu;
Roof2StatusWord.7   := GVL_Roof.IRiegel22auf;
Roof2StatusWord.8   := GVL_Roof.IDach2Schnell;


(*** MQTT Section ***)
MQTTTimer(IN:=TRUE);
IF MQTTTimer.Q OR Roof1Status <> LastRoof1Status OR Roof2Status <> LastRoof2Status THEN
	MQTTClient.Publish('roof', 'roof1', 'Roof1Status', RoofStatus_TO_String(Roof1Status, Quoted := TRUE));
	MQTTClient.Publish('roof', 'roof2', 'Roof2Status', RoofStatus_TO_String(Roof2Status, Quoted := TRUE));
	MQTTClient.Publish('environment', 'weatherstation', 'WeatherBad',	BOOL_TO_STRING(EnvironmentAlarm));		
	MQTTClient.Publish('roof', 'main', 'isRoofManual',	BOOL_TO_STRING(isRoofManual));		
	MQTTClient.Publish('roof', 'roof1', 'Roof1StatusWord',	WORD_TO_STRING(Roof1StatusWord));		
	MQTTClient.Publish('roof', 'roof2', 'Roof2StatusWord',	WORD_TO_STRING(Roof2StatusWord));		
	
	MQTTTimer(IN:=FALSE);
	LastRoof1Status := Roof1Status;
	LastRoof2Status := Roof2Status;
END_IF

END_PROGRAM

// ---- POUs/Function Blocks/FB_RoofControl.TcPOU
FUNCTION_BLOCK FB_RoofControl
VAR_INPUT
	cmdRoofCommand:	E_RoofCommand;
	bLocked1:    	BOOL;  // Riegel11zu
	bUnlocked1:  	BOOL;  // Riegel11auf
	bLocked2:    	BOOL;  // Riegel21zu
	bUnlocked2:  	BOOL;  // Riegel21auf
  	bFastSwitch:    BOOL;  // Dach1schnell
	bOpenSwitch1:	BOOL;  // Dach1auf
	bOpenSwitch2:	BOOL;  // Dach1auf2
	bClosedSwitch1:	BOOL;  // Dach1zu
	bClosedSwitch2:	BOOL;  // Dach1zu2
END_VAR
VAR_OUTPUT
	bOpenLock1:		BOOL;	// Riegel11auf
	bCloseLock1:	BOOL;	// Riegel11zu
	bOpenLock2:		BOOL;	// Riegel21auf
	bCloseLock2:	BOOL;	// Riegel21zu
	bRoofOpen:		BOOL;	// Dach1auf
	bRoofClose:		BOOL;	// Dach1zu
	bMotorFast:		BOOL;	// Dach1schnell 
	RoofStatus:		E_RoofStatus := StatusUndefined;
	MotionAlarm:	BOOL;	
END_VAR
VAR
	// new status of the roof
	nStatus:			E_RoofStatus;
	// both locks engaged
	isBothLocked:		BOOL;
	// both locks open
	isBothUnlocked:		BOOL;
	// one lock engaged
	isOneLocked:		BOOL;
	// one lock open
	isOneUnlocked:		BOOL;
	// roof is closed
	isClosed:			BOOL;
	// on limit switch reports closed
	isOneClosed:		BOOL;
	// roof is open
	isOpen:				BOOL;
	isMotorFast:		BOOL;
	RoofOpenDelayed,
	RoofCloseDelayed,
	MotorFastDelayed: 	BOOL;
	OpenDelay:			TON;
	CloseDelay:			TON;
	FastDelay:			TON;
	isClosedDelay:		TON;
	F_Closed,
	F_Fast,
	F_Open:			F_TRIG;
	R_Fast:			R_TRIG;
	lastError:			E_ErrorFlag;
END_VAR

(* open_roof_command or close_roof_command may change state immediatly *)
nStatus := StatusUndefined;

// Helper variables
isOneLocked := bLocked1 OR bLocked2;
isOneUnlocked := bUnlocked1 OR bUnlocked2;
isBothLocked := bLocked1 AND bLocked2; 
isBothUnlocked := bUnlocked1 AND bUnlocked2;
isOneClosed := bClosedSwitch1 OR bClosedSwitch2;
isClosedDelay(IN := bClosedSwitch1 OR bClosedSwitch2, PT := T#4S, Q => isClosed);
isOpen:= bOpenSwitch1 OR bOpenSwitch2;
isMotorFast := (NOT bFastSwitch); 


// Generic conditions
IF isOpen THEN bRoofOpen := FALSE; END_IF
IF isClosed THEN bRoofClose := FALSE; END_IF
IF bRoofClose THEN bRoofOpen := FALSE; END_IF
MotorFastDelayed := isMotorFast; 
// IF bUnlocked1 THEN bOpenLock1 := FALSE; END_IF
// IF bUnlocked2 THEN bOpenLock2 := FALSE; END_IF
IF bCloseLock1 THEN bOpenLock1 := FALSE; END_IF
IF bCloseLock2 THEN	bOpenLock2 := FALSE; END_IF

IF bLocked1 THEN bCloseLock1 := FALSE; END_IF
IF bLocked2 THEN bCloseLock2 := FALSE; END_IF


// detect falling edge of closed switch
F_Closed(CLK := isClosed);
F_Fast(CLK := isMotorFast);
R_Fast(CLK := isMotorFast);
F_Open(CLK := isOpen);


IF cmdRoofCommand = OpenRoof THEN
	// OpenRoof Conditions
	bCloseLock1 := FALSE;
	bCloseLock2 := FALSE;
	IF NOT bUnlocked1 AND NOT bCloseLock1 THEN bOpenLock1 := TRUE; END_IF
	IF NOT bUnlocked2 AND NOT bCloseLock2 THEN bOpenLock2 := TRUE; END_IF
	RoofCloseDelayed  := FALSE;
	RoofOpenDelayed := isBothUnlocked AND NOT isOpen AND NOT bRoofClose;	
	//RoofOpenDelayed := isOneUnlocked AND NOT isOpen AND NOT bRoofClose;	
	
	// identify OpenRoof States
	IF bOpenLock1 OR bOpenLock2 THEN nStatus := StatusUnlocking; END_IF
	IF F_Closed.Q THEN nStatus := StatusStartOpening; END_IF
	IF isMotorFast THEN nStatus := StatusOpening; END_IF
	IF F_Fast.Q THEN nStatus := StatusEndOpening; END_IF
	// guess status based on the previous one
	IF nStatus = StatusEndClosing THEN nStatus := StatusStartOpening; END_IF
	IF nStatus = StatusStartClosing THEN nStatus := StatusEndOpening; END_IF
	
ELSIF cmdRoofCommand = CloseRoof THEN
	// CloseRoof Conditions
	bOpenLock1 := NOT isClosed AND NOT bUnlocked1;
	bOpenLock2 := NOT isClosed AND NOT bUnlocked2;
	bCloseLock1 := isClosed AND NOT isOpen AND NOT bLocked1 AND NOT bOpenLock1;
	bCloseLock2 := isClosed AND NOT isOpen AND NOT bLocked2 AND NOT bOpenLock2;
	RoofOpenDelayed := FALSE;
	RoofCloseDelayed := isBothUnlocked AND NOT isOneLocked AND NOT isCLosed AND NOT bRoofOpen;
	//RoofCloseDelayed := isOneUnlocked AND NOT isOneLocked AND NOT isCLosed AND NOT bRoofOpen;

	// identify CloseRoof States
	IF bCloseLock1 OR bCloseLock2 THEN nStatus := StatusLocking; END_IF
	IF F_Open.Q THEN nStatus := StatusStartClosing; END_IF
	IF isMotorFast THEN nStatus := StatusClosing; END_IF
	IF F_Fast.Q THEN nStatus := StatusEndClosing; END_IF
	// guess status based on the previous one
	IF nStatus = StatusStartOpening THEN nStatus := StatusEndClosing; END_IF
	IF nStatus = StatusEndOpening THEN nStatus := StatusStartClosing; END_IF

ELSE // Stop the Roof
	bCloseLock1 := FALSE;
	bCloseLock2 := FALSE;
	bOpenLock1 := FALSE;
	bOpenLock2 := FALSE;
	bRoofOpen := FALSE;
	bRoofClose := FALSE;
	bMotorFast := FALSE;
	RoofOpenDelayed := FALSE;
	RoofCloseDelayed := FALSE;
	MotorFastDelayed := FALSE; 
	
	// stopped Roof States
	//IF NOT isOpen AND NOT isOneClosed THEN nStatus := StatusUndefined; END_IF

END_IF

// generic States:
IF isOneClosed THEN
	IF isBothUnlocked THEN
		nStatus := StatusClosed;
	END_IF
	IF isBothLocked THEN
		nStatus := StatusLocked;
	END_IF
END_IF
IF isOpen THEN
	nStatus := StatusOpened;
END_IF
IF isOpen AND isClosed THEN
	nStatus := StatusError;
	lastError := E_ErrorFlag.ErrorOpenClose;
END_IF
// if roof is open and is Locked
IF (NOT isOneClosed) AND isOneLocked THEN
	nStatus := StatusError;
	lastError := E_ErrorFlag.ErrorOpenLocked;
END_IF
// if one of the locks is locked and unlocked at the same time
IF (bLocked1 AND bUnlocked1) OR (bLocked2 AND bUnlocked2) THEN
	nStatus := StatusError;
	lastError := E_ErrorFlag.ErrorLockUnlock;
END_IF

OpenDelay(IN := RoofOpenDelayed, PT := T#4S, Q => bRoofOpen);
CloseDelay(IN := RoofCloseDelayed, PT := T#4S, Q => bRoofClose);
FastDelay(IN := MotorFastDelayed AND (bRoofOpen OR bRoofClose), PT := T#2S, Q => bMotorFast);

MotionAlarm := 	(RoofOpenDelayed AND NOT bRoofOpen) OR
				(RoofCloseDelayed AND NOT bRoofClose);

// Statemachine for operation
(*
IF nStatus = StatusError THEN
	bCloseLock1 := FALSE;
	bCloseLock2 := FALSE;
	bOpenLock1 := FALSE;
	bOpenLock2 := FALSE;
	bRoofOpen := FALSE;
	bRoofClose := FALSE;
	bMotorFast := FALSE;
	RoofOpenDelayed := FALSE;
	RoofCloseDelayed := FALSE;
	MotorFastDelayed := FALSE;
	
END_IF


*)
RoofStatus := nStatus;

END_FUNCTION_BLOCK

// ---- POUs/Function Blocks/LIGHT_BUTTON.TcPOU
FUNCTION_BLOCK LIGHT_BUTTON
VAR_INPUT
	IN:	BOOL;
	PT: TIME := T#1H;
END_VAR
VAR_OUTPUT
	Q: BOOL;
	Q1: BOOL;
END_VAR
VAR
	onstate:	BOOL;
	trigger:	R_TRIG;
	// main timer
	lighttimer: TP;
	// first warning pulse
	pulse1:	TP;
	// second warning pulse
	pulse2: TP;
	// third warning pulse
	pulse3: TP;
	pulse1delay: TON;
	pulse2delay: TON;
	pulse3delay: TON;
END_VAR

trigger(CLK := IN);
IF trigger.Q THEN // if we detect a button press, we flip the onstate
	onstate := NOT onstate;
END_IF
lighttimer(IN := onstate, PT := PT);
pulse1delay(IN:= lighttimer.Q, PT := PT - T#20S);
pulse1(IN := pulse1delay.Q, PT := T#250MS);
pulse2delay(IN:= lighttimer.Q, PT := PT - T#10S);
pulse2(IN := pulse2delay.Q, PT := T#250MS);
pulse3delay(IN:= lighttimer.Q, PT := PT - T#10S + T#500MS);
pulse3(IN := pulse3delay.Q, PT := T#250MS);

Q := onstate AND lighttimer.Q AND NOT pulse1.Q AND NOT pulse2.Q AND NOT pulse3.Q;
Q1 := onstate AND lighttimer.Q;
IF NOT Q1 THEN
	onstate := FALSE;
END_IF

END_FUNCTION_BLOCK

// ---- POUs/Function Blocks/FB_StatusLamp.TcPOU
FUNCTION_BLOCK FB_StatusLamp
VAR_INPUT
	RoofStatus: E_RoofStatus;
END_VAR
VAR_OUTPUT
	RoofLamp: BOOL;
END_VAR
VAR
	LampPause: TIME := T#10S;
	Blink:			FB_BLINK;
END_VAR

IF RoofStatus = StatusError THEN 
	LampPause := T#1S;
ELSIF RoofStatus = StatusUndefined THEN 
	LampPause := T#3S;
ELSE
	LampPause := T#10S;
	RoofLamp := FALSE;
END_IF;
Blink(ENABLE := (RoofStatus = StatusError) OR (RoofStatus = StatusUndefined), 
		ON_TIME := T#1S,
		OFF_TIME := LampPause,
		Q => RoofLamp);

END_FUNCTION_BLOCK

// ---- POUs/Function Blocks/FB_BLINK.TcPOU
FUNCTION_BLOCK FB_BLINK
VAR_INPUT
	ENABLE:		BOOL;
	ON_TIME:	TIME := T#1S;
	OFF_TIME:	TIME := T#3S;
END_VAR
VAR_OUTPUT
	Q:		BOOL;
END_VAR
VAR
    IMPULS   :TOF;
    PAUSE    :TOF;
END_VAR

IMPULS(IN:= NOT PAUSE.Q AND NOT IMPULS.Q, PT:= ON_TIME);
PAUSE(IN:= NOT PAUSE.Q AND NOT IMPULS.Q, PT:= OFF_TIME);
Q := IMPULS.Q AND ENABLE;

END_FUNCTION_BLOCK

// ---- POUs/Function Blocks/FB_MQTTCommunication.TcPOU
FUNCTION_BLOCK FB_MQTTCommunication
VAR_INPUT
END_VAR
VAR_OUTPUT
END_VAR
VAR
	GetHostName:		FB_GetHostName;
	HostName: 			STRING(255);
    bSetParameter:		BOOL := FALSE;
    bConnect:			BOOL := FALSE;
    (* received message *)
	bSubscribed: 		BOOL;
	sTopicSub: 			STRING(255) := 'STELLA/Telemetry/SET';
	{attribute 'TcEncoding':='UTF-8'}
	sTopicRcv: 			STRING(255);
	{attribute 'TcEncoding':='UTF-8'}
	fbMessageQueue:		FB_IotMqttMessageQueue;
    fbMessage:			FB_IotMqttMessage;
	fbMqttClient:		FB_IotMqttClient;
	sPayloadRcv: 		STRING;
	influxMessage:		InfluxMessage;
	measurement, 
	parameter, 
	value:		STRING(255);
END_VAR

(*
MQTT Communication section

Source:
https://infosys.beckhoff.com/english.php?content=../content/1033/tf6701_tc3_iot_communication_mqtt/3518541195.html&id=

*)
IF HostName='' THEN
	GetHostName.bExecute := TRUE;
ELSE
	GetHostName.bExecute := FALSE;
	bSetParameter := TRUE;
END_IF

GetHostName(sHostName => HostName);

// set the parameters once
IF bSetParameter THEN
    bSetParameter               := FALSE;
    fbMqttClient.sHostName      := '161.72.132.74'; //'192.168.1.74';
    fbMqttClient.nHostPort      := 1883;
    fbMqttClient.sClientId      := HostName; 
    fbMqttClient.sTopicPrefix   := ''; 
	fbMqttClient.nKeepAlive     := 60; 
    fbMqttClient.ipMessageQueue := fbMessageQueue;
	bConnect := TRUE;
END_IF

// connect to the client
IF NOT fbMqttClient.bConnected THEN
;
END_IF

fbMqttClient.Execute(bConnect);
	
IF fbMqttClient.bConnected THEN
    IF NOT bSubscribed THEN
        bSubscribed := fbMqttClient.Subscribe(sTopic:=sTopicSub, 
												eQoS:=TcIotMqttQos.AtMostOnceDelivery);
    END_IF
END_IF

// receive queued messages
IF fbMessageQueue.nQueuedMessages > 0 THEN
    IF fbMessageQueue.Dequeue(fbMessage:=fbMessage) THEN
        fbMessage.GetTopic(pTopic:=ADR(sTopicRcv), nTopicSize:=SIZEOF(sTopicRcv) );
        fbMessage.GetPayload(pPayload:=ADR(sPayloadRcv), nPayloadSize:=SIZEOF(sPayloadRcv), bSetNullTermination:=TRUE);
		ADSLOGSTR( ADSLOG_MSGTYPE_HINT OR ADSLOG_MSGTYPE_LOG, 'MQTT %s', sPayloadRcv);
		IF sTopicRcv = sTopicSub THEN
			influxMessage(  sPayload := sPayloadRcv, measurement => measurement, parameter => parameter, value => value);
			IF measurement = 'command' THEN
				IF parameter = 'OpenRoofAuto' THEN
					MAIN.OpenRoofAuto := STRING_TO_BOOL(value);
				ELSIF parameter = 'CloseRoofAuto' THEN
					MAIN.CloseRoofAuto := STRING_TO_BOOL(value);
				ELSIF parameter = 'StopRoofAuto' THEN
					MAIN.StopRoofAuto := STRING_TO_BOOL(value);
				ELSIF parameter = 'LightAuto' THEN
					MAIN.LightAuto := STRING_TO_BOOL(value);
				ELSIF parameter = 'RoofPower' THEN
					Auxiliary.RoofPower := STRING_TO_BOOL(value);
				ELSIF parameter = 'Dehumidifier' THEN
					DehumidifierControl.ManualEnable := STRING_TO_BOOL(value);
				ELSIF parameter = 'ThAr1' THEN
					CalibrationUnit.lampindex := 1;
					CalibrationUnit.lampenable := STRING_TO_BOOL(value);
				ELSIF parameter = 'ThAr2' THEN
					CalibrationUnit.lampindex := 2;
					CalibrationUnit.lampenable := STRING_TO_BOOL(value);
				ELSIF parameter = 'Halo1' THEN
					CalibrationUnit.lampindex := 3;
					CalibrationUnit.lampenable := STRING_TO_BOOL(value);
				ELSIF parameter = 'Halo2' THEN
					CalibrationUnit.lampindex := 4;
					CalibrationUnit.lampenable := STRING_TO_BOOL(value);
				END_IF // parameter
			END_IF // measurement
		END_IF // Topic
		sPayloadRcv := '';
    END_IF // Dequeue
END_IF

PROPERTY Error : BOOL
GET
Error := fbMqttClient.bError;
END_GET
END_PROPERTY

METHOD Publish : BOOL
VAR_INPUT
	domain: 	STRING(255) := 'environment';
	location: 	STRING(255) := 'roof';
	parameter:	STRING(255);
	value:		STRING(255);
END_VAR
VAR
	sPayloadPub: STRING(255) := '';
	fbFormat:	FB_FormatString;
	bError:		BOOL;
	nErrID: UDINT;
	retain_message:		BOOL := FALSE;
END_VAR
//sPayloadPub := 'environment,location=roof,host=CX-4E6032 ';
fbFormat( sFormat := '%s,location=%s,host=%s %s=%s', 
			arg1 := F_STRING(domain), 
			arg2 := F_STRING(location), 
			arg3 := F_STRING(HostName),
			arg4 := F_STRING(parameter),
			arg5 := F_STRING(value),
 
			sOut => sPayloadPub,
			bError => bError, 
			nErrID => nErrID );
// retain message if value is boolean
retain_message := value = 'TRUE' OR value = 'FALSE';

Publish := fbMqttClient.Publish(	
				sTopic:= 'STELLA/Telemetry', 
				pPayload:= ADR(sPayloadPub), 
				nPayloadSize:= LEN2(ADR(sPayloadPub)),
				eQoS:= TcIotMqttQos.AtMostOnceDelivery,
				bRetain:= retain_message, 
				bQueue:= FALSE );
END_METHOD

METHOD PublishLog : BOOL
VAR_INPUT
	level: 	STRING(255) := 'INFO';
	message:	STRING(255);
	
END_VAR
VAR
	sPayloadPub: STRING(255) := '';
	fbFormat:	FB_FormatString;
	bError:		BOOL;
	nErrID: UDINT;
END_VAR
VAR_OUTPUT
	published: BOOL;
END_VAR
//sPayloadPub := 'environment,location=roof,host=CX-4E6032 ';
fbFormat( sFormat := 'log,host=%s,level=%s message="%s"', 
			arg1 := F_STRING(HostName), 
			arg2 := F_STRING(level), 
			arg3 := F_STRING(message),
 
			sOut => sPayloadPub,
			bError => bError, 
			nErrID => nErrID );

published := fbMqttClient.Publish(	
				sTopic:= 'STELLA/Log', 
				pPayload:= ADR(sPayloadPub), 
				nPayloadSize:= LEN2(ADR(sPayloadPub)),
				eQoS:= TcIotMqttQos.AtMostOnceDelivery,
				bRetain:= FALSE, 
				bQueue:= FALSE );
END_METHOD

END_FUNCTION_BLOCK

// ---- POUs/Auxiliary.TcPOU
PROGRAM Auxiliary
VAR_INPUT
	RoofPower:	BOOL;
END_VAR
VAR
	MS1NC1,
	MS2NC1,
	MS3NC1,
	MS4NC1,
	MS5NC1,
	MS6NC1:	BOOL;

	MS1NC2,
	MS2NC2,
	MS3NC2,
	MS4NC2,
	MS5NC2,
	MS6NC2:	BOOL;

	NC1Status: WORD;
	LastNC1Status: WORD := 16#FFFF;
	
	NC2Status: WORD;
	LastNC2Status: WORD := 16#FFFF;
END_VAR

GVL_Environment.RoofPower := RoofPower;

MS1NC1 := NOT GVL_Roof.IMotorschutz11;
MS2NC1 := NOT GVL_Roof.IMotorschutz12;
MS3NC1 := NOT GVL_Roof.IMotorschutz13;
MS4NC1 := NOT GVL_Roof.IMotorschutz14;
MS5NC1 := NOT GVL_Roof.IMotorschutz15;
MS6NC1 := NOT GVL_Roof.IMotorschutz16;

MS1NC2 := NOT GVL_Roof.IMotorschutz21;
MS2NC2 := NOT GVL_Roof.IMotorschutz22;
MS3NC2 := NOT GVL_Roof.IMotorschutz23;
MS4NC2 := NOT GVL_Roof.IMotorschutz24;
MS5NC2 := NOT GVL_Roof.IMotorschutz25;
MS6NC2 := NOT GVL_Roof.IMotorschutz26;

NC1Status.0 := MS1NC1;
NC1Status.1 := MS2NC1;
NC1Status.2 := MS3NC1;
NC1Status.3 := MS4NC1;
NC1Status.4 := MS5NC1;
NC1Status.5 := MS6NC1;

IF NC1Status <> LastNc1Status THEN
	MAIN.MQTTClient.Publish('roof', 'roof1', 'NC1Status', WORD_TO_STRING(NC1Status));
	LastNc1Status := NC1Status;
END_IF

NC2Status.0 := MS1NC2;
NC2Status.1 := MS2NC2;
NC2Status.2 := MS3NC2;
NC2Status.3 := MS4NC2;
NC2Status.4 := MS5NC2;
NC2Status.5 := MS6NC2;

IF NC2Status <> LastNc2Status THEN
	MAIN.MQTTClient.Publish('roof', 'roof2', 'NC2Status', WORD_TO_STRING(NC2Status));
	LastNc2Status := NC2Status;
END_IF

END_PROGRAM

// ---- POUs/DehumidifierControl.TcPOU
PROGRAM DehumidifierControl
VAR_INPUT
	// enable signal for der Dehumidifier
	Enable:	BOOL := TRUE;
	// manual enable signal
	ManualEnable: BOOL;
END_VAR
VAR
	// run dehumidifer at last for n seconds to avoid fast switching cycles
	HumidityTrigger: SR;
	RunDelay : TON := (PT:=T#30S);
	ManualTimer: TON := (PT := T#3H);
	LowOverride: TON := (PT := T#3H);
	// classic event log
	DehumidifierLog: FB_EventLog;
	
	OnTrigger:	R_TRIG;
	OffTrigger:	F_TRIG;
END_VAR
VAR CONSTANT
	HumidityBayLow:		REAL := 65.0;
	HumidityBayHigh:	REAL := 75.0;
END_VAR

HumidityTrigger( SET1 := ManualEnable OR 
						LowOverride.Q OR
						(Enable AND Environment.HumidityBay > HumidityBayHigh),
				RESET := Environment.HumidityBay < HumidityBayLow);
// override if we stay above low limit for too long
LowOverride( In := Environment.HumidityBay > HumidityBayLow);
				
// deactivate Manual Signal aftern n hours
ManualTimer( IN := ManualEnable);
IF ManualTimer.Q AND ManualEnable THEN
	ManualEnable := FALSE;
END_IF

// delay switch on to avoid overload
RunDelay(IN := HumidityTrigger.Q1);
GVL_Environment.Dehumidifier := RunDelay.Q;

DehumidifierLog(Trigger := GVL_Environment.Dehumidifier, OnMessage := 'The dehumidifier is on.', OffMessage := 'The dehumidifier is off.');

(*** MQTT Section ***)
OnTrigger(CLK := GVL_Environment.Dehumidifier);
OffTrigger(CLK := GVL_Environment.Dehumidifier);
IF OnTrigger.Q OR OffTrigger.Q THEN
	MAIN.MQTTClient.Publish('bay', 'bay', 'Dehumidifier', BOOL_TO_STRING(GVL_Environment.Dehumidifier));
END_IF

END_PROGRAM

// ---- POUs/Function Blocks/FB_EventLog.TcPOU
FUNCTION_BLOCK FB_EventLog
VAR_INPUT
	Trigger:		BOOL;
	// ADSLOG_MSGTYPE_HINT or ADSLOG_MSGTYPE_WARN or ADSLOG_MSGTYPE_ERROR
	Level:			UDINT := ADSLOG_MSGTYPE_HINT;
	FormatString: 	STRING(255) := '%s';
	OnMessage: 		STRING(255) := '';
	OffMessage:		STRING(255) := '';
	OffLevel:		UDINT := ADSLOG_MSGTYPE_HINT;
END_VAR
VAR_OUTPUT
END_VAR
VAR
	LogonTrigger: R_TRIG;
	LogoffTrigger: F_TRIG;
	PayloadMessage: STRING(255);
	fbFormat:	FB_FormatString;
	LevelString: STRING;
END_VAR

LogonTrigger(CLK := Trigger);
LogoffTrigger(CLK := Trigger);
// in case the OffLevel is not set use the default Level Value
IF OffLevel = 0 THEN
	OffLevel := Level;
END_IF
IF LogonTrigger.Q AND LEN(OnMessage)>0 THEN
	ADSLOGSTR( Level OR ADSLOG_MSGTYPE_LOG, FormatString, OnMessage);
END_IF

IF LogoffTrigger.Q AND LEN(OffMessage)>0 THEN
	ADSLOGSTR( OffLevel OR ADSLOG_MSGTYPE_LOG, FormatString, OffMessage);
END_IF

IF LogonTrigger.Q AND LEN(OnMessage)>1 THEN
	IF Level=ADSLOG_MSGTYPE_HINT THEN
		LevelString := 'INFO';
	ELSIF Level=ADSLOG_MSGTYPE_WARN THEN
		LevelString := 'WARNING';
	ELSE
	    LevelString := 'ERROR';
	END_IF
	fbFormat( sFormat := FormatString, arg1 := F_STRING(OnMessage), sOut => PayloadMessage);
	MAIN.MQTTClient.PublishLog(LevelString, PayloadMessage);

END_IF

IF LogoffTrigger.Q AND LEN(OffMessage)>1 THEN
	IF OffLevel=ADSLOG_MSGTYPE_HINT THEN
		LevelString := 'INFO';
	ELSIF OffLevel=ADSLOG_MSGTYPE_WARN THEN
		LevelString := 'WARNING';
	ELSE
	    LevelString := 'ERROR';
	END_IF
	fbFormat( sFormat := FormatString, arg1 := F_STRING(OffMessage), sOut => PayloadMessage);
	MAIN.MQTTClient.PublishLog(LevelString, PayloadMessage);
END_IF

END_FUNCTION_BLOCK

// ---- POUs/Environment.TcPOU
PROGRAM Environment
VAR
	LightDirection:	REAL;
	Brightness1:	REAL;
	WindSpeed1:		REAL;
	Temperature1:	REAL;
	Humidity1:		REAL;
	Rain_analogue1:	REAL;
	WindDirection:	REAL;
	Pressure0, Pressure:		REAL;
	
	WindSpeed2:		REAL;
	Temperature2:	REAL;
	Humidity2:		REAL;
	Brightness2:		REAL;
	WindSpeed:		REAL;
	Humidity:		REAL;
	// electronics room temperature
	Temperature_Electronics:	REAL;
	// electronics room humidity
	Humidity_Electronics:		REAL;
	// telescope bay temperature
	TemperatureBay:	REAL;
	// telescope bay humidity
	HumidityBay:	REAL;
	// SES Spectrograph temperature
	Temperature_Spec:	REAL;
	// SES spectrograph humidity
	Humidity_Spec:		REAL;
	// wind speed at bay
	Windspeed_bay:		REAL;
	// old pressure sensor from weather station 1 (West)
	Pressure_bay:		REAL;
	// analog dust sensor
	
	Dust:				REAL;
	// digital rain sensor
	RainAlarm1:			BOOL;
	// digital rain sensor
	RainAlarm2:			BOOL;
	// combination of rain sensors
	RainMasterAlarm:	BOOL;
	// delay timer for digital rain signal 1
	RainTimer1:			TON;
	// delay timer for digital rain signal 2
	RainTimer2:			TON;
	// delay timer for combined rain signals
	RainMasterTimer:	TON;
	Rain1_brokendelay:	TON := (PT := T#60M);
	Humidity1_brokendelay:	TON := (PT := T#480M);
	Humidity2_brokendelay:	TON := (PT := T#480M);
	Wind1_brokendelay:	TON := (PT := T#60M);
	Wind2_brokendelay:	TON := (PT := T#60M);
	// maximum wind speed 1
	MaximumWind1: REAL;
	MaximumWind2: REAL;
	DustAvg:	FB_TimeAverage;
	WindAvg1:	FB_TimeAverage; 
	Windavg2:	FB_TimeAverage;
	PressureAverage:	FB_TimeAverage;
	// Dust Sensors
	DigitalDust1:	FB_Dust;
	DigitalDust2:	FB_Dust;
	Dust11Kalman:	FB_Kalman1D;
	Dust12Kalman:	FB_Kalman1D;
	Dust21Kalman:	FB_Kalman1D;
	Dust22Kalman:	FB_Kalman1D;
	dustratio:		LREAL := 1.0;
	// Kalman Process noise variance
	Qv_Kalman:		LREAL := 1E-5;
	// Kalman measurement noise variance
	Vv_Kalman:		LREAL := 1E-3;
	// Triggers
	ElectronicsTemperatureTrigger:	SR;
	ElectronicsHumidityTrigger:		SR;
	SpectrographTemperatureTrigger:	SR;
	SpectrographHumidityTrigger:	SR;
	EnvironmentHumidityTrigger:		SR;
	BayHumidityTrigger:				SR;
	BayHumidityCriticalTrigger:		SR;
	DustTrigger:					SR;
	Rainanalogue1brokenTrigger:		SR;
	Rainanalogue2brokenTrigger:		SR;
	// MQTT timer
	MQTTTimer : TON := (PT:=T#5S);
END_VAR
VAR_OUTPUT
	Rain_analogue1_broken:	BOOL;
	Rain_analogue2_broken:	BOOL;
	Humidity1_broken:		BOOL;
	Humidity2_broken:		BOOL;
	Wind1_broken:			BOOL;
	Wind2_broken:			BOOL;
	Dust_broken:			BOOL;
END_VAR
VAR CONSTANT
	h:	REAL := 2390.0;
END_VAR

(* convert raw Sensor values to real values *)
(* Weather Station 1 *)
LightDirection := 	F_Y(GVL_Environment.rawLightDirection,	0, 32767,	0.0, 360.0); // degrees
Brightness1 := 		F_Y(GVL_Environment.rawBrightness,		0, 32767,	0.0, 120000.0); // Lux
Pressure0 := 		F_Y(GVL_Environment.rawPressure,		0, 32767,	800.0, 1020.0); // hPa
Humidity1 :=		F_Y(GVL_Environment.rawHumidity1, 		16, 32767,   0.0, 100.0); // %
Temperature1 :=  	F_Y(GVL_Environment.rawTemperature1, 	0, 32767, -40.0, 60.0); // °C
Rain_analogue1 := 	F_Y(GVL_Environment.rawRain_analogue1,	8, 32767,	0.0, 100.0); // mm/h
WindDirection := 	F_Y(GVL_Environment.rawWindDirection,	0, 32767,   0.0, 360.0); // degrees
WindSpeed1 := 		F_Y(GVL_Environment.rawWindSpeed1, 		0, 32767,   0.0, 60.0); // m/s

Pressure := LREAL_TO_REAL(Pressure0 * EXPT(1.0 - (0.0065*h/(Temperature1+273.15)) , 5.255));

RainAlarm1 := Rain_analogue1 > 0.5; // was 0.1
RainAlarm2 := NOT GVL_Environment.Rain_alarm2;

RainTimer1(IN := RainAlarm1, PT := T#30S);
RainTimer2(IN := RainAlarm2, PT := T#30S);
RainMasterTimer(IN := RainAlarm1 AND RainAlarm2, PT := T#5S);
RainMasterAlarm := RainTimer1.Q OR RainTimer2.Q OR RainMasterTimer.Q;


(*  Weather Station 2 *)

WindSpeed2 := 		F_Y(GVL_Environment.rawWindSpeed2, 		0, 32767,   0.0, 50.0); // m/s
Temperature2 :=  	F_Y(GVL_Environment.rawTemperature2, 	0, 32767, -30.0, 70.0); // °C
Humidity2 :=		F_Y(GVL_Environment.rawHumidity2, 		0, 32767,   0.0, 100.0); // %

Brightness2 :=		F_Y(GVL_Environment.rawBrightness, 		0, 32767,   0.0, 150000.0); // lux
IF Brightness2 < 1000.0 THEN 
	Brightness2 :=	F_Y(GVL_Environment.rawBrightnessLow, 	0, 32767,   0.000, 1000.0); // lux
END_IF


(* Indoor environment *)

Temperature_Electronics :=  F_Y(GVL_Environment.rawTemperature_Electronics, 	0, 32767, -30.0, 70.0); // °C
Humidity_Electronics :=		F_Y(GVL_Environment.rawHumidity_Electronics, 		0, 32767,   0.0, 100.0); // %
TemperatureBay :=  			F_Y(GVL_Environment.rawTemperatureBay, 				0, 32767, -30.0, 70.0); // °C
HumidityBay := 				F_Y(GVL_Environment.rawHumidityBay, 				0, 32767,   0.0, 100.0); // %
Temperature_Spec :=  		F_Y(GVL_Environment.rawTemperature_Spec, 			0, 32767, -30.0, 70.0); // °C
Humidity_Spec := 			F_Y(GVL_Environment.rawHumidity_Spec, 				0, 32767,   0.0, 100.0); // %
Windspeed_bay := 			F_Y(GVL_Environment.rawWindSpeedBay, 				0, 32767,   0.0, 40.0); // m/s
Pressure_bay := 			F_Y(GVL_Environment.rawPressureBay,					0, 16383,	600.0, 1060.0); // hPa 0..5V -> 600...1060hPa

WindAvg1(IN := WindSpeed1, PT := T#2M, MAXAVG=> MaximumWind1);
WindAvg2(IN := WindSpeed2, PT := T#2M, MAXAVG=> MaximumWind2);
PressureAverage(IN := Pressure, PT := T#1M);
WindSpeed := MAX(WindSpeed1, WindSpeed2);
Humidity := MAX(Humidity1, Humidity2);

ElectronicsTemperatureTrigger(SET1 := Temperature_Electronics >= 30.0, RESET := Temperature_Electronics < 25.0);
SpectrographTemperatureTrigger(SET1 := Temperature_Spec >= 30.0, RESET := Temperature_Spec < 25.0);
ElectronicsHumidityTrigger(SET1 := Humidity_Electronics >= 65.0, RESET := Humidity_Electronics < 50.0);
SpectrographHumidityTrigger(SET1 := Humidity_Spec >= 65.0, RESET := Humidity_Spec < 50.0);
EnvironmentHumidityTrigger(SET1 := Humidity >= MAIN.HumidityLimitHigh, RESET := HumidityBay < MAIN.HumidityLimitLow);
BayHumidityTrigger(SET1 := HumidityBay >= MAIN.HumidityLimitHigh, RESET := HumidityBay < MAIN.HumidityLimitLow);
BayHumidityCriticalTrigger(SET1 := HumidityBay >= MAIN.HumidityLimitCritical, RESET := HumidityBay < MAIN.HumidityLimitHigh);

Rainanalogue1brokenTrigger( SET1:= RainMasterAlarm AND Rain_analogue1 < 1E-3, RESET := Rain_analogue1 > 1E-2);
Rain1_brokendelay( IN := Rainanalogue1brokenTrigger.Q1);
Humidity1_brokendelay(IN := Humidity > 10.0 AND Humidity1 < 0.5 * Humidity);
Humidity2_brokendelay(IN := Humidity > 10.0 AND Humidity2 < 0.5 * Humidity);
Humidity1_broken:= Humidity1_brokendelay.Q;
Humidity2_broken:= Humidity2_brokendelay.Q;
Wind1_brokendelay(IN := WindSpeed1 < 0.5 * WindSpeed);
Wind1_broken:= Wind1_brokendelay.Q;
Wind2_brokendelay(IN := WindSpeed2 < 0.5 * WindSpeed);
Wind2_broken:= Wind2_brokendelay.Q;

(*** Dust section ***)
// digital dust sensors
DigitalDust1(pwm1 := GVL_Environment.rawDust11, pwm2 := GVL_Environment.rawDust12);
DigitalDust2(pwm1 := GVL_Environment.rawDust21, pwm2 := GVL_Environment.rawDust22);
Dust11Kalman(z := dustratio * DigitalDust1.concentration1 / 1000.0, Q := Qv_Kalman, V := Vv_Kalman);
Dust12Kalman(z := dustratio * DigitalDust1.concentration2 / 1000.0, Q := Qv_Kalman, V := Vv_Kalman);
Dust21Kalman(z := dustratio * DigitalDust2.concentration1 / 1000.0, Q := Qv_Kalman, V := Vv_Kalman);
Dust22Kalman(z := dustratio * DigitalDust2.concentration2 / 1000.0, Q := Qv_Kalman, V := Vv_Kalman);


Dust_broken := (GVL_Environment.rawDust = 0) OR (GVL_Environment.rawDust >= 32000);
Dust := F_Y(GVL_Environment.rawDust, 0, 32767,   0.0, 0.1);
IF Dust_broken THEN
	Dust := dustratio * DigitalDust1.concentration2 / 1000.0;
END_IF
DustAvg(IN := Dust, PT := T#2M); // m^3
DustTrigger( SET1 := DustAvg.AVG > 0.01, RESET := DustAvg.AVG < 0.0075);

(* MQTT Section *)

MQTTTimer(IN:=TRUE);
IF MQTTTimer.Q THEN // publish new payload every second
	
	MAIN.MQTTClient.Publish('environment', 'weatherstation1', 'EnvironmentLightDirection',	LREAL_TO_FMTSTR(LightDirection, 2, TRUE));
	MAIN.MQTTClient.Publish('environment', 'weatherstation1', 'EnvironmentBrightness1',		LREAL_TO_FMTSTR(Brightness1, 2, TRUE));		
	MAIN.MQTTClient.Publish('environment', 'weatherstation1', 'EnvironmentWindSpeed1',		LREAL_TO_FMTSTR(WindSpeed1, 2, TRUE));		
	MAIN.MQTTClient.Publish('environment', 'weatherstation1', 'EnvironmentTemperature1',	LREAL_TO_FMTSTR(Temperature1, 2, TRUE));
	IF Humidity1 > 1.0 THEN
		MAIN.MQTTClient.Publish('environment', 'weatherstation1', 'EnvironmentHumidity1',		LREAL_TO_FMTSTR(Humidity1, 2, TRUE));		
	END_IF
	MAIN.MQTTClient.Publish('environment', 'weatherstation1', 'EnvironmentRain1',			LREAL_TO_FMTSTR(Rain_analogue1, 5, TRUE));		
	MAIN.MQTTClient.Publish('environment', 'weatherstation1', 'EnvironmentWindDirection',	LREAL_TO_FMTSTR(WindDirection, 1, TRUE));		
	MAIN.MQTTClient.Publish('environment', 'weatherstation1', 'EnvironmentPressure',		LREAL_TO_FMTSTR(PressureAverage.AVG, 2, TRUE));		
	MAIN.MQTTClient.Publish('environment', 'weatherstation1', 'EnvironmentRainAlarm1',		BOOL_TO_STRING(RainAlarm1));		
	
	MAIN.MQTTClient.Publish('environment', 'weatherstation2', 'EnvironmentTemperature2',LREAL_TO_FMTSTR(Temperature2, 2, TRUE));
	MAIN.MQTTClient.Publish('environment', 'weatherstation2', 'EnvironmentHumidity2', 	LREAL_TO_FMTSTR(Humidity2, 2, TRUE));		
	MAIN.MQTTClient.Publish('environment', 'weatherstation2', 'EnvironmentWindSpeed2', 	LREAL_TO_FMTSTR(WindSpeed2, 2, TRUE));		
	MAIN.MQTTClient.Publish('environment', 'weatherstation2', 'EnvironmentBrightness2',	LREAL_TO_FMTSTR(Brightness2, 2, TRUE));		
	MAIN.MQTTClient.Publish('environment', 'weatherstation2', 'EnvironmentDust',		LREAL_TO_FMTSTR(Dust, 5, TRUE));		
	MAIN.MQTTClient.Publish('environment', 'weatherstation2', 'EnvironmentRainAlarm2',	BOOL_TO_STRING(RainAlarm2));		
	
	MAIN.MQTTClient.Publish('environment', 'base', 'ElectronicsTemperature',	LREAL_TO_FMTSTR(Temperature_Electronics, 2, TRUE));
	MAIN.MQTTClient.Publish('environment', 'base', 'ElectronicsHumidity',		LREAL_TO_FMTSTR(Humidity_Electronics, 2, TRUE));		
	
	MAIN.MQTTClient.Publish('environment', 'bay', 'BayTemperature',	LREAL_TO_FMTSTR(TemperatureBay, 2, TRUE));
	MAIN.MQTTClient.Publish('environment', 'bay', 'BayHumidity',	LREAL_TO_FMTSTR(HumidityBay, 2, TRUE));		
	MAIN.MQTTClient.Publish('environment', 'bay', 'BayWindSpeed',	LREAL_TO_FMTSTR(Windspeed_bay, 2, TRUE));		
	MAIN.MQTTClient.Publish('environment', 'bay', 'BayPressure',	LREAL_TO_FMTSTR(Pressure_bay, 2, TRUE));		
	
	MAIN.MQTTClient.Publish('environment', 'weatherstation', 'EnvironmentDustPM1',	LREAL_TO_FMTSTR(Dust11Kalman.x, 5, TRUE));		
	MAIN.MQTTClient.Publish('environment', 'weatherstation', 'EnvironmentDustPM25',	LREAL_TO_FMTSTR(Dust12Kalman.x, 5, TRUE));		
	
	MAIN.MQTTClient.Publish('environment', 'bay', 'EnvironmentDust2PM1',	LREAL_TO_FMTSTR(Dust21Kalman.x, 5, TRUE));		
	MAIN.MQTTClient.Publish('environment', 'bay', 'EnvironmentDust2PM25',	LREAL_TO_FMTSTR(Dust22Kalman.x, 5, TRUE));		
	
	MAIN.MQTTClient.Publish('environment', 'spectrograph', 'SpectrographTemperature',	LREAL_TO_FMTSTR(Temperature_Spec, 2, TRUE));
	MAIN.MQTTClient.Publish('environment', 'spectrograph', 'SpectrographHumidity',		LREAL_TO_FMTSTR(Humidity_Spec, 2, TRUE));		
	MQTTTimer(IN:=FALSE);	
END_IF

END_PROGRAM

// ---- POUs/Function Blocks/FB_Kalman1D.TcPOU
FUNCTION_BLOCK FB_Kalman1D
VAR_INPUT
	// Measurement input
	z: LREAL;
END_VAR
VAR_IN_OUT
	// Process noise variance
    Q:	LREAL;  
	// Measurement noise variance
    V:	LREAL;   
END_VAR
VAR_OUTPUT
	// Kalman gain
	K: LREAL;
	// Filtered state
	x: LREAL;
END_VAR
VAR
	// Error covariance
	P: LREAL := 1.0;
	// State estimate
	x_est: LREAL := 0.0;
END_VAR

// Kalman Filter Execution
P := P + Q;  // Prediction covariance
K := P / (P + V); // Kalman gain
x_est := x_est + K * (z - x_est); // Update estimate
P := (1 - K) * P; // Update covariance
x := x_est;

END_FUNCTION_BLOCK

// ---- POUs/Functions/F_Y.TcPOU
FUNCTION F_Y : REAL
VAR_INPUT
	fX:		REAL;
	fXmin, fXmax:	REAL;
	fYmin, fYmax:	REAL;
END_VAR
VAR
	fgain,
	foffset:	REAL;
END_VAR

(*
y = mx+b

		    delta X	  fYmax - fYmin
m = fgain = ------- = -------------
			delta Y	  fXmax - fXmin
			
b = foffset = y - m*x = y - fgain*x
					  = fYmin - fgain * fXmin
*)

// y = fgain * x + foffset

IF (fXmax - fXmin) <> 0 THEN

	// Berechnung der Steigung
	fgain := (fYmax - fYmin) / (fXmax - fXmin);
	
	// Berechnung des Offsets
	foffset := fYmin - (fgain * fXmin);
	
	// Berechnung von F_Y

	IF fgain * fX + foffset < fYmin THEN 
		F_Y := fYmin;
		
	END_IF
	IF fgain * fX + foffset > fYmax THEN 
		F_Y := fYmax;
	END_IF	
	F_Y := fgain * fX + foffset;
	F_Y := LIMIT(fYmin, F_Y, FYmax);	
END_IF

END_FUNCTION

// ---- POUs/CalibrationUnit.TcPOU
PROGRAM CalibrationUnit
VAR_INPUT
	lampindex: USINT;
	lampenable:	BOOL;
END_VAR
VAR
	lampsensor1	AT%I*: BOOL;
	lampsensor2	AT%I*: BOOL;
	ThArlamp1	AT%Q*: BOOL;
	ThArlamp2	AT%Q*: BOOL;
	Halolamp1	AT%Q*: BOOL;
	Halolamp2	AT%Q*: BOOL;
	
	SESdewarpressureraw 	AT%I*:	INT;
	SESpumppressureraw 		AT%I*:	INT;
	cryosupplyraw 	AT%I*:	INT;
	cryoreturnraw	 AT%I*:	INT;
	
	rawTemperature1	AT%I*:	INT;
	rawTemperature2	AT%I*:	INT;
	rawTemperature3	AT%I*:	INT;
	rawTemperature4	AT%I*:	INT;
	rawTemperature5	AT%I*:	INT;
	rawTemperature6	AT%I*:	INT;
	// volts
	SESdewarvoltage:	REAL;
	// volts
	SESpumpvoltage:		REAL;
// MQTT timer
	MQTTTimer : TON := (PT:=T#5S);
END_VAR
VAR_OUTPUT
	// mbar
	SESdewarpressure: 	REAL;
	// mbar
	SESpumppressure: 	REAL;
	// Bar
	cryosupply: 	REAL;
	// Bar
	cryoreturn: 	REAL;
	
	temperature1: 	REAL;
	temperature2: 	REAL;
	temperature3: 	REAL;
	temperature4: 	REAL;
	temperature5: 	REAL;
	temperature6: 	REAL;
	meantemperature:	REAL;
END_VAR

SESdewarvoltage :=	F_Y(SESdewarpressureraw, 	0, 32767,   0.0, 10.0);
SESpumpvoltage :=	F_Y(SESpumppressureraw, 	0, 32767,   0.0, 10.0);
SESdewarpressure := LREAL_TO_REAL(EXPT(10.0, 1.667 * SESdewarvoltage - 17.07691)); // d = 11.33
SESpumppressure  := LREAL_TO_REAL(EXPT(10.0, F_Y(SESpumpvoltage, 2.0, 10.0, -9.0, 3.0)));

cryosupply := 		F_Y(cryosupplyraw, 		0, 32767,   0.0, 25.0);
cryoreturn := 		F_Y(cryoreturnraw, 		0, 32767,   0.0, 25.0);

temperature1 := rawTemperature1 / 100.0;
temperature2 := rawTemperature2 / 100.0;
temperature3 := rawTemperature3 / 100.0;
temperature4 := rawTemperature4 / 100.0;
temperature5 := rawTemperature5 / 100.0;
temperature6 := rawTemperature6 / 100.0;

CASE lampindex OF
	1:	ThArlamp1 := lampenable;
		ThArlamp2 := FALSE;
		Halolamp1 := FALSE;
		Halolamp2 := FALSE;
		
	2:	ThArlamp1 := FALSE;
		ThArlamp2 := lampenable;
		Halolamp1 := FALSE;
		Halolamp2 := FALSE;
		
	3:	ThArlamp1 := FALSE;
		ThArlamp2 := FALSE;
		Halolamp1 := lampenable;
		Halolamp2 := FALSE;
		
	4:	ThArlamp1 := FALSE;
		ThArlamp2 := FALSE;
		Halolamp1 := FALSE;
		Halolamp2 := lampenable;
ELSE
	ThArlamp1 := FALSE;
	ThArlamp2 := FALSE;
	Halolamp1 := FALSE;
	Halolamp2 := FALSE;
	lampenable := FALSE;
END_CASE

MQTTTimer(IN:=TRUE);
IF MQTTTimer.Q THEN // publish new payload every second
	MAIN.MQTTClient.Publish('environment', 'calibrationunit', 'thar1on',	BOOL_TO_STRING(NOT lampsensor1));
	MAIN.MQTTClient.Publish('environment', 'calibrationunit', 'thar2on',	BOOL_TO_STRING(NOT lampsensor2));
	MAIN.MQTTClient.Publish('environment', 'calibrationunit', 'oil1_temperature',	LREAL_TO_FMTSTR(temperature1, 2, TRUE));
	MAIN.MQTTClient.Publish('environment', 'calibrationunit', 'oilroom1_temperature',	LREAL_TO_FMTSTR(temperature2, 2, TRUE));
	MAIN.MQTTClient.Publish('environment', 'calibrationunit', 'oil2_temperature',	LREAL_TO_FMTSTR(temperature3, 2, TRUE));
	MAIN.MQTTClient.Publish('environment', 'calibrationunit', 'oilroom2_temperature',	LREAL_TO_FMTSTR(temperature4, 2, TRUE));
	MAIN.MQTTClient.Publish('environment', 'calibrationunit', 'lounge_temperature',	LREAL_TO_FMTSTR(temperature5, 2, TRUE));
	MAIN.MQTTClient.Publish('environment', 'calibrationunit', 'lab_temperature',	LREAL_TO_FMTSTR(temperature6, 2, TRUE));
	MAIN.MQTTClient.Publish('environment', 'calibrationunit', 'CryoPressureSupply',	REAL_TO_STRING(cryosupply));
	MAIN.MQTTClient.Publish('environment', 'calibrationunit', 'CryoPressureReturn',	REAL_TO_STRING(cryoreturn));
	MAIN.MQTTClient.Publish('environment', 'calibrationunit', 'SESDewarPressure',	REAL_TO_STRING(SESdewarpressure));
	MAIN.MQTTClient.Publish('environment', 'calibrationunit', 'SESpumpPressure',	REAL_TO_STRING(SESpumppressure));
	
END_IF

END_PROGRAM

// ---- POUs/Function Blocks/TIMER.TcPOU
FUNCTION_BLOCK TIMER
VAR_INPUT
	bStart : BOOL := TRUE;
END_VAR
VAR_OUTPUT
	tDifference : TIME;
END_VAR
VAR
	tTimeReturn1:	TIME;
	tTimeReturn2:	TIME;
	fbTrigger1:		R_TRIG;
	fbTrigger2:		F_TRIG;
END_VAR

fbTrigger1(CLK := bStart);
fbTrigger2(CLK := bStart);

IF fbTrigger1.Q THEN
	tTimeReturn1 := TIME();
END_IF

IF bStart OR fbTrigger2.Q THEN
	tTimeReturn2 := TIME();
END_IF

tDifference := tTimeReturn2 - tTimeReturn1;

END_FUNCTION_BLOCK

// ---- POUs/Chamber.TcPOU
PROGRAM Chamber
VAR
	// SES cover(=copy of room regulation)
	rawTemperature1	AT%I*:	INT;
	// inside SES cover
	rawTemperature2	AT%I*:	INT;
	// optical bench inside of cover
	rawTemperature3	AT%I*:	INT;
	// floor(copy of floor regulation)
	rawTemperature4	AT%I*:	INT;
	//optical bench outside cover
	rawTemperature5	AT%I*:	INT;
	// e-box
	rawTemperature6	AT%I*:	INT;
	// pressure sensor 4mA...20mA => 700mbar ... 900mbar
	rawpressure 	AT%I*:	INT;
	// MQTT timer
	MQTTTimer : TON := (PT:=T#5S);
END_VAR
VAR_OUTPUT
	// SES cover(=copy of room regulation)
	temperature1: 	REAL;
	// inside SES cover
	temperature2: 	REAL;
	// optical bench inside of cover
	temperature3: 	REAL;
	// floor(copy of floor regulation)
	temperature4: 	REAL;
	//optical bench outside cover
	temperature5: 	REAL;
	// e-box
	temperature6: 	REAL;
	// average temperature
	chambertemperature:	REAL;
	// mbar
	chamberpressure: 	REAL;
END_VAR

temperature1 := rawTemperature1 / 100.0;
temperature2 := rawTemperature2 / 100.0;
temperature3 := rawTemperature3 / 100.0;
temperature4 := rawTemperature4 / 100.0;
temperature5 := rawTemperature5 / 100.0;
temperature6 := rawTemperature6 / 100.0;

chambertemperature := (	temperature2 +
						temperature3 +
						temperature4 +
						temperature5) / 4.0;
						

chamberpressure :=	F_Y(rawpressure, 	0, 32767,   700.0, 900.0);

MQTTTimer(IN:=TRUE);
IF MQTTTimer.Q THEN // publish new payload every second
	MAIN.MQTTClient.Publish('environment', 'chamber', 'temperature1',	LREAL_TO_FMTSTR(temperature1, 2, TRUE));
	MAIN.MQTTClient.Publish('environment', 'chamber', 'temperature2',	LREAL_TO_FMTSTR(temperature2, 2, TRUE));
	MAIN.MQTTClient.Publish('environment', 'chamber', 'temperature3',	LREAL_TO_FMTSTR(temperature3, 2, TRUE));
	MAIN.MQTTClient.Publish('environment', 'chamber', 'temperature4',	LREAL_TO_FMTSTR(temperature4, 2, TRUE));
	MAIN.MQTTClient.Publish('environment', 'chamber', 'temperature5',	LREAL_TO_FMTSTR(temperature5, 2, TRUE));
	MAIN.MQTTClient.Publish('environment', 'chamber', 'temperature6',	LREAL_TO_FMTSTR(temperature6, 2, TRUE));
	MAIN.MQTTClient.Publish('environment', 'chamber', 'chamber_temperature',	REAL_TO_STRING(chambertemperature));
	MAIN.MQTTClient.Publish('environment', 'chamber', 'chamber_pressure',	REAL_TO_STRING(chamberpressure));
END_IF

END_PROGRAM

// ---- POUs/Logging.TcPOU
PROGRAM Logging
VAR
	// Logging voriables
	EnvironmentLog,
	DustLog,
	HumidityLog,
	HumidityErrorLog,
	HumidityBayLog,
	WindSpeedLog,
	WindSpeedBayLog,
	Rain1Log,
	Rain2Log,
	OpenRoof1Log, CloseRoof1Log, StopRoof1Log,
	OpenRoof2Log, CloseRoof2Log, StopRoof2Log,
	Roof1StatusLog, Roof2StatusLog,
	Roof1ErrorLog, Roof2ErrorLog,
	Roof1WarningLog, Roof2WarningLog,
	LightLog,
	ManualLog,
	RoofOpenLog,
	RoofUnlockedLog,
	RoofClosedLog: FB_EventLog;
	
	ElectronicsTemperatureLog,
	ElectronicsHumidityLog,
	SpectrographTemperatureLog,
	SpectrographHumidityLog,
	UsUndervoltageLog,
	UpUndervoltageLog,
	MotorProtection1Log,
	MotorProtection2Log: FB_EventLog;
	
	RoofOpenTimeoutLog,
	RoofCloseTimeoutLog,
	Roof1LockTimeoutLog,
	Roof2LockTimeoutLog,
	Roof1UnlockTimeoutLog,
	Roof2UnlockTimeoutLog:	FB_EventLog;
	
	Rain_analogue1_brokenLog,
	Rain_analogue2_brokenLog,
	Humidity1_brokenLog,
	Humidity2_brokenLog,
	Wind1_brokenLog,
	Wind2_brokenLog,
	Dust_brokenLog:	FB_EventLog;
	
	
	LastRoof1Status,
	LastRoof2Status:	E_RoofStatus;

END_VAR

(*** Logging Section ***)

EnvironmentLog(	Trigger := MAIN.EnvironmentAlarm AND (MAIN.Roof1Status = StatusOpened), 
				Level := ADSLOG_MSGTYPE_WARN, OnMessage := 'The weather is bad!', OffMessage := 'The weather is good.');
DustLog(		Trigger := Environment.DustTrigger.Q1 AND (MAIN.Roof1Status = StatusOpened), 
				Level := ADSLOG_MSGTYPE_WARN, OnMessage := 'Dust is over limit!');
HumidityLog(	Trigger := Main.HumidityTrigger.Q1 AND (MAIN.Roof1Status = StatusOpened), Level := ADSLOG_MSGTYPE_WARN, OnMessage := 'Humidity is over limit!');
HumidityErrorLog(	Trigger := Environment.HumidityBay > 85.0, Level := ADSLOG_MSGTYPE_ERROR, OnMessage := 'Bay humidity is high! Dehumidifier failure!');
HumidityBayLog(	Trigger := Environment.BayHumidityTrigger.Q1, Level := ADSLOG_MSGTYPE_WARN, 
				OnMessage := 'Bay humidity bay is over limit', 
				OffMessage := 'Bay humidity is nominal.');
WindSpeedLog(	Trigger := Environment.WindSpeed > MAIN.WindSpeedLimit AND (MAIN.Roof1Status = StatusOpened), 
				Level := ADSLOG_MSGTYPE_WARN, OnMessage := 'Wind speed is over limit!');
WindSpeedBayLog(Trigger := Environment.Windspeed_bay > MAIN.WindSpeedBayLimit, Level := ADSLOG_MSGTYPE_WARN, OnMessage := 'Wind speed in bay is over limit');
// Rain1Log(		Trigger := NOT GVL_Environment.Rain_alarm1, Level := ADSLOG_MSGTYPE_WARN, OnMessage := 'Rain alarm 1 is on!');
// Rain2Log(		Trigger := NOT GVL_Environment.Rain_alarm2, Level := ADSLOG_MSGTYPE_WARN, OnMessage := 'Rain alarm 2 is on!');

OpenRoof1Log( Trigger := MAIN.Roof1Command = OpenRoof, OnMessage := 'Open roof 1');
OpenRoof2Log( Trigger := MAIN.Roof2Command = OpenRoof, OnMessage := 'Open roof 2');
CloseRoof1Log( Trigger := MAIN.Roof1Command = CloseRoof, OnMessage := 'Close roof 1');
CloseRoof2Log( Trigger := MAIN.Roof2Command = CloseRoof, OnMessage := 'Close roof 2');
StopRoof1Log( Trigger := MAIN.Roof1Command = StopRoof, OnMessage := 'Stop roof 1');
StopRoof2Log( Trigger := MAIN.Roof2Command = StopRoof, OnMessage := 'Stop roof 2');

Roof1ErrorLog( Trigger := MAIN.Roof1Status = StatusError, Level := ADSLOG_MSGTYPE_ERROR, OnMessage := 'Roof 1 has an error!');
Roof2ErrorLog( Trigger := MAIN.Roof2Status = StatusError, Level := ADSLOG_MSGTYPE_ERROR, OnMessage := 'Roof 2 has an error!');

Roof1WarningLog( Trigger := MAIN.Roof1Status = StatusUndefined, Level := ADSLOG_MSGTYPE_WARN, OnMessage := 'The status of roof 1 is undefined!');
Roof2WarningLog( Trigger := MAIN.Roof2Status = StatusUndefined, Level := ADSLOG_MSGTYPE_WARN, OnMessage := 'The status of roof 2 is undefined!');

//Roof1StatusLog( Trigger :=  MAIN.Roof1Status <> LastRoof1Status, FormatString := 'Roof1 status: %s', OnMessage := RoofStatus_TO_String(Main.Roof1Status, Quoted := FALSE));
//Roof2StatusLog( Trigger :=  MAIN.Roof2Status <> LastRoof2Status, FormatString := 'Roof2 status: %s', OnMessage := RoofStatus_TO_String(Main.Roof2Status, Quoted := FALSE));
LastRoof1Status := MAIN.Roof1Status;
LastRoof2Status := MAIN.Roof2Status;

RoofOpenLog( Trigger := (MAIN.Roof1Status = StatusOpened) OR (MAIN.Roof2Status = StatusOpened), Level := ADSLOG_MSGTYPE_WARN, OnMessage := 'The roof is open.');
RoofUnlockedLog( Trigger := (MAIN.Roof1Status = StatusUnlocked) OR (MAIN.Roof2Status = StatusUnlocked), 
					Level := ADSLOG_MSGTYPE_WARN, OnMessage := 'The roof is unlocked.');
RoofClosedLog( Trigger := (MAIN.Roof1Status = StatusLocked) AND (MAIN.Roof2Status = StatusLocked), 
				OnMessage := 'The roof is closed and locked.');

LightLog(Trigger := GVL_Environment.LightSwitch, Level := ADSLOG_MSGTYPE_WARN, OnMessage := 'The light is on manually.', OffMessage := 'The light is off.');
ManualLog(Trigger := MAIN.isRoofManual, Level := ADSLOG_MSGTYPE_WARN, OnMessage := 'Roof is in manual mode.', OffMessage := 'Roof is in automatic mode.');

ElectronicsTemperatureLog( Trigger := Environment.ElectronicsTemperatureTrigger.Q1 , 
							Level := ADSLOG_MSGTYPE_ERROR, 
							OnMessage := 'Electronics temperature is over limit!');

ElectronicsHumidityLog( Trigger := Environment.ElectronicsHumidityTrigger.Q1 , 
							Level := ADSLOG_MSGTYPE_ERROR, 
							OnMessage := 'Electronics humidity is over limit!');

SpectrographTemperatureLog( Trigger := Environment.SpectrographTemperatureTrigger.Q1 , 
							Level := ADSLOG_MSGTYPE_ERROR, 
							OnMessage := 'Spectrograph temperature is over limit!');

SpectrographHumidityLog( Trigger := Environment.SpectrographHumidityTrigger.Q1 , 
							Level := ADSLOG_MSGTYPE_ERROR, 
							OnMessage := 'Spectrograph humidity is over limit!');
UsUndervoltageLog( Trigger := GVL_Panel.Us_Undervoltage, 
							Level := ADSLOG_MSGTYPE_ERROR, 
							OnMessage := 'Us undervoltage!');
UpUndervoltageLog( Trigger := GVL_Panel.Up_Undervoltage, 
							Level := ADSLOG_MSGTYPE_ERROR, 
							OnMessage := 'Up undervoltage! / EMERGENCY STOP!');
MotorProtection1Log( Trigger := Auxiliary.NC1Status <> 0, 
							Level := ADSLOG_MSGTYPE_ERROR, 
							OnMessage := 'Roof1 motor protection fault!');
MotorProtection2Log( Trigger := Auxiliary.NC2Status <> 0, 
							Level := ADSLOG_MSGTYPE_ERROR, 
							OnMessage := 'Roof2 motor protection fault!');
							
RoofOpenTimeoutLog( Trigger := MAIN.Roof1OpenTimeOut.Q OR MAIN.Roof2OpenTimeOut.Q, Level := ADSLOG_MSGTYPE_ERROR, OnMessage := 'Roof time out error while opening!');
RoofCloseTimeoutLog( Trigger := MAIN.Roof1CloseTimeOut.Q OR MAIN.Roof2CloseTimeOut.Q, Level := ADSLOG_MSGTYPE_ERROR, OnMessage := 'Roof timeout error while closing!');

Roof1LockTimeoutLog( Trigger := MAIN.Roof1LockTimeOut.Q, Level := ADSLOG_MSGTYPE_ERROR, OnMessage := 'Roof1 lock time out!');
Roof2LockTimeoutLog( Trigger := MAIN.Roof2LockTimeOut.Q, Level := ADSLOG_MSGTYPE_ERROR, OnMessage := 'Roof2 lock time out!');
Roof1UnlockTimeoutLog( Trigger := MAIN.Roof1UnlockTimeOut.Q, Level := ADSLOG_MSGTYPE_ERROR, OnMessage := 'Roof1 unlock time out!');
Roof2UnlockTimeoutLog( Trigger := MAIN.Roof2UnlockTimeOut.Q, Level := ADSLOG_MSGTYPE_ERROR, OnMessage := 'Roof2 unlock time out!');

Rain_analogue1_brokenLog( Trigger := Environment.Rain1_brokendelay.Q, Level := ADSLOG_MSGTYPE_WARN, OnMessage := 'Analog rain sensor 1 signal implausble!');
Rain_analogue2_brokenLog( Trigger := Environment.Rainanalogue2brokenTrigger.Q1, Level := ADSLOG_MSGTYPE_WARN, OnMessage := 'Analog rain sensor 2 signal implausble!');
Humidity1_brokenLog( Trigger := Environment.Humidity1_broken, Level := ADSLOG_MSGTYPE_WARN, OnMessage := 'Humidity sensor 1 signal implausble!');
Humidity2_brokenLog( Trigger := Environment.Humidity2_broken, Level := ADSLOG_MSGTYPE_WARN, OnMessage := 'Humidity sensor 2 signal implausible!');
Wind1_brokenLog( Trigger := Environment.Wind1_broken, Level := ADSLOG_MSGTYPE_WARN, OnMessage := 'Wind sensor 1 signal implausble!');
Wind2_brokenLog( Trigger := Environment.Wind2_broken, Level := ADSLOG_MSGTYPE_WARN, OnMessage := 'Wind sensor 2 signal implausble!');
Dust_brokenLog( Trigger := Environment.Dust_broken, Level := ADSLOG_MSGTYPE_ERROR, OnMessage := 'Analogue dust sensor is broken! Fail-over to digital sensor.');

END_PROGRAM

// ---- POUs/Functions/RoofStatus_TO_String.TcPOU
FUNCTION RoofStatus_TO_String : STRING
VAR_INPUT
	RoofStatus: E_RoofStatus;
	Quoted: BOOL := FALSE;
END_VAR
VAR
	result:	STRING(15);
END_VAR

(*
	StatusUndefined 	:= 0,
	StatusClosed 		:= 100,
	StatusLocking 		:= 200,
	StatusLocked 		:= 300,
	StatusUnlocking 	:= 400,
	StatusUnlocked 		:= 500,
	StatusStartOpening 	:= 600,
	StatusOpening 		:= 700,
	StatusEndOpening 	:= 800,
	StatusOpened 		:= 900,
	StatusStartClosing 	:= 1000,
	StatusClosing 		:= 1100,
	StatusEndClosing 	:= 1200,
	
	StatusError 		:= -1

*)
IF RoofStatus = StatusError THEN
	result := 'Error';
ELSIF RoofStatus = StatusClosed THEN
	result := 'Closed';
ELSIF RoofStatus = StatusLocking THEN
	result := 'Locking';
ELSIF RoofStatus = StatusLocked THEN
	result := 'Locked';
ELSIF RoofStatus = StatusUnlocking THEN
	result := 'Unlocking';
ELSIF RoofStatus = StatusUnlocked THEN
	result := 'Unlocked';
ELSIF RoofStatus = StatusStartOpening THEN
	result := 'StartOpening';
ELSIF RoofStatus = StatusOpening THEN
	result := 'Opening';
ELSIF RoofStatus = StatusEndOpening THEN
	result := 'EndOpening';
ELSIF RoofStatus = StatusOpened THEN
	result := 'Opened';
ELSIF RoofStatus = StatusStartClosing THEN
	result := 'StartClosing';
ELSIF RoofStatus = StatusClosing THEN
	result := 'Closing';
ELSIF RoofStatus = StatusEndClosing THEN
	result := 'EndClosing';
ELSE
	result := 'Undefined';
END_IF

IF Quoted THEN
	result := CONCAT('"', result);
	RoofStatus_TO_String := CONCAT(result ,'"');
ELSE
	RoofStatus_TO_String := result;
END_IF

END_FUNCTION

// ---- POUs/Function Blocks/FB_PRECESS3.TcPOU
FUNCTION_BLOCK FB_PRECESS3
VAR_INPUT
	// right ascension in degrees
	ra: LREAL;
	// declination in degrees
	dec: LREAL;
	
END_VAR
VAR_OUTPUT
	// precessed right ascension
	ra_precessed:	LREAL;
	// precessed declination
	dec_precessed:	LREAL;
END_VAR
VAR
	ra_rad, dec_rad: LREAL;
	// starting jd (J2000)
	jd0: LREAL;
	// traget JD
	jd: LREAL;
	t, 
	eta, 
	z, 
	phi,
	A,
	B,
	C	: LREAL;
END_VAR
VAR CONSTANT
	deg_to_rad : LREAL := PI/180.0;
	sec_to_rad : LREAL := deg_to_rad/3600.0;
END_VAR

// see Jean Meeus p.135

ra_rad := ra*deg_to_rad;
dec_rad := dec*deg_to_rad;

// todo epoch to jd and jd0
JD := MAIN.jd;
jd0 := 2451545.0;
t := (jd - jd0) / 36525.0;

eta :=	(2306.2181*t + 0.30188*t*t + 0.017998*t*t*t) * sec_to_rad;
z :=	(2306.2181*t + 1.09468*t*t + 0.018203*t*t*t) * sec_to_rad;
phi :=	(2004.3109*t - 0.42665*t*t - 0.041833*t*t*t) * sec_to_rad;

A :=            COS(dec_rad) * SIN(ra_rad + eta);
B := COS(phi) * COS(dec_rad) * COS(ra_rad + eta) - SIN(phi) * SIN(dec_rad);
C := SIN(phi) * COS(dec_rad) * COS(ra_rad + eta) + COS(phi) * SIN(dec_rad);

// tan(ra - z) == A/B
ra_precessed := MODABS((ATAN2(A, B) + z)/deg_to_rad, 360);
IF ABS(dec) > 89.5 THEN
	dec_precessed := ACOS(SQRT(A*A + B*B))/deg_to_rad;
ELSE
	// sin(de)c = C
	dec_precessed := ASIN(C)/deg_to_rad;	
END_IF

END_FUNCTION_BLOCK
